// TwinCAT 3 PLC project PLC1
// Title: Sample Demo-Rack
// Company: Beckhoff Automation GmbH & Co. KG
// Author: Michael Golz
// ProjectVersion: 1.0.0
// ProgramVersion: 3.1.4026.26
// libraries:
//   Standard, * (System)
//   Tc2_Drive, * (Beckhoff Automation GmbH)
//   Tc2_EtherCAT, * (Beckhoff Automation GmbH)
//   Tc2_IoFunctions, * (Beckhoff Automation GmbH)
//   Tc2_Math, * (Beckhoff Automation GmbH)
//   Tc2_MC2, * (Beckhoff Automation GmbH)
//   Tc2_MC2_Camming, * (Beckhoff Automation GmbH)
//   Tc2_MC2_Drive, * (Beckhoff Automation GmbH)
//   Tc2_MC2_XFC, * (Beckhoff Automation GmbH)
//   Tc2_NCI, * (Beckhoff Automation GmbH)
//   Tc2_NcKinematicTransformation, * (Beckhoff Automation GmbH)
//   Tc2_PlcInterpolation, * (Beckhoff Automation GmbH)
//   Tc2_Standard, * (Beckhoff Automation GmbH)
//   Tc2_SUPS, * (Beckhoff Automation GmbH)
//   Tc2_System, * (Beckhoff Automation GmbH)
//   Tc2_Utilities, * (Beckhoff Automation GmbH)
//   Tc3_Database, * (Beckhoff Automation GmbH)
//   Tc3_EventLogger, * (Beckhoff Automation GmbH)
//   Tc3_Interfaces, * (Beckhoff Automation GmbH)
//   Tc3_IotBase, * (Beckhoff Automation GmbH)
//   Tc3_JsonXml, * (Beckhoff Automation GmbH)
//   Tc3_Mc3Base, * (Beckhoff Automation GmbH)
//   Tc3_Mc3FluidPower, * (Beckhoff Automation GmbH)
//   Tc3_Mc3Ptp, * (Beckhoff Automation GmbH)
//   Tc3_Module, * (Beckhoff Automation GmbH)
//   Tc3_RealtimeMonitoring, * (Beckhoff Automation GmbH)
//   TwinSafe3Diagnostics_v0.2.3, * (Beckhoff Automation LLC - Sample Code)
//   VisuDialogs, * (System)
// project tree:
//   DUTs/00_MainBlocks/ E_SystemStartupSequence.TcDUT (not stored)
//   DUTs/20_Axis/ E_AxisReversingSequence.TcDUT (not stored), E_McResetStatus.TcDUT (not stored)
//   DUTs/30_EtherCatDiagnostic/ E_EcDiacStatus.TcDUT (not stored), E_EcGetSlaveName.TcDUT (not stored), E_EcSystemStatus.TcDUT (not stored), ST_EcTerminalDiagInfo.TcDUT (not stored)
//   DUTs/40_TwinSAFE/ ST_AdsAddr.TcDUT (not stored)
//   DUTs/40_TwinSAFE/TwinSAFE_Connection/AX5805/ E_TsDiagnosisObjektsFA10AX5805.TcDUT (not stored), E_TsErrIndicesFA82AX5805.TcDUT (not stored), ST_TsControlWordAX5805.TcDUT (not stored), ST_TsDiagObjectsFA10AX5805.TcDUT (not stored), ST_TsErrIndicesFA82AX5805.TcDUT (not stored), ST_TsStatusWordAX5805.TcDUT (not stored)
//   DUTs/40_TwinSAFE/TwinSAFE_Connection/EK1914/ ST_TsDiagObjectsBitsEK1914.TcDUT (not stored), ST_TsDiagObjectsEK1914.TcDUT (not stored)
//   DUTs/40_TwinSAFE/TwinSAFE_Connection/EL1904/ ST_TsDiagObjectsBitsEL1904.TcDUT (not stored), ST_TsDiagObjectsEL1904.TcDUT (not stored)
//   DUTs/40_TwinSAFE/TwinSAFE_Connection/EL2904/ ST_TsDiagObjectsBitsEL2904.TcDUT (not stored), ST_TsDiagObjectsEL2904.TcDUT (not stored)
//   DUTs/40_TwinSAFE/TwinSAFE_Connection/ E_TsCycleDiagObj.TcDUT (not stored), ST_TsConnectionInfo1Byte.TcDUT (not stored), ST_TsConnectionInfo2Byte.TcDUT (not stored), ST_TsConnectionInfo8Byte.TcDUT (not stored), ST_TsConnectionInfoEL3214.TcDUT (not stored), ST_TsConnectionInfoEL5021.TcDUT (not stored), ST_TsSlave2Temp.TcDUT (not stored), ST_TsSlave3Temp.TcDUT (not stored)
//   DUTs/40_TwinSAFE/TwinSAFE_Functionblocks/ E_TsFbType.TcDUT (not stored), ST_TsFbInfo.TcDUT (not stored)
//   DUTs/40_TwinSAFE/TwinSAFE_Group/ ST_TsGroupInfo.TcDUT (not stored)
//   DUTs/ E_SampleMode.TcDUT (not stored)
//   / extMarkTask.TcTTO (not stored), FluidPowerSim.TcTTO, GlobalTextList.TcGTLO (not stored), NC_Task_1_SAF.TcTTO, PlcTask.TcTTO, PlcTaskFast.TcTTO (not stored), Visualization Manager.TcVMO (not stored)
//   GVLs/ GVL.TcGVL, GVL00_IO_CX.TcGVL (not stored), GVL01_IO_EK1100.TcGVL (not stored), GVL02_IO_EK1101.TcGVL (not stored), GVL10_VAR_PRG.TcGVL (not stored), GVL20_Axis.TcGVL, GVL30_DiagnosticEtherCAT.TcGVL (not stored)
//   POUs/MC3/ExternalSetpoint_Mc3_Nc2/ ExtSetpoint_MC3_NC2.TcPOU, FB_ExtSg_FollowNcAxis.TcPOU, PRG_SAF.TcPOU
//   POUs/MC3/ExternalSetpoint_Mc3_Nc2/Support/ E_Command.TcDUT, E_State.TcDUT
//   POUs/MC3/Gearing/ MC3_Gearing.TcPOU
//   POUs/MC3/Gearing/Support/ CompareLREAL.TcPOU, E_Axis.TcDUT, E_GearCommand.TcDUT, NextMinorStep.TcPOU (not stored), NextStep.TcPOU (not stored), SetStep.TcPOU
//   POUs/MC3/LoadControl/ LoadControl.TcPOU, LoadControlSim.TcPOU
//   POUs/MC3/PressToTarget/ PressToTarget.TcPOU, PressToTargetSim.TcPOU
//   POUs/MC3/ReversingSequence/ MC3_ReversingSequence.TcPOU
//   POUs/Motion/ CamTable.TcPOU (not stored), Ext_SP_Gen.TcPOU (not stored), Axis1.TcPOU, AxisGeneral.TcPOU (not stored), Axis2.TcPOU, Axis3.TcPOU, Axis4.TcPOU, NCI.TcPOU (not stored)
//   POUs/Database Server/ CSVSample.TcPOU (not stored), E_WriteMode.TcDUT (not stored), FB_CSV_Access.TcPOU (not stored), ST_CSVDataStruct.TcDUT (not stored)
//   POUs/GeneralPlcBlocks/ FB_GenerateData.TcPOU (not stored), Blinker.TcPOU (not stored), ClockGenerator.TcPOU (not stored), GeneralPlc.TcPOU (not stored)
//   POUs/IoT and JsonXml/FBs/ FB_JSONEncoding.TcPOU (not stored), FB_MqttCom_String.TcPOU (not stored), prgPopulateStructure.TcPOU (not stored)
//   POUs/IoT and JsonXml/ IoTDataStruct.TcDUT (not stored), IoT_JSON_XML.TcPOU (not stored)
//   POUs/MainPOUs/ MAIN.TcPOU, MAINFast.TcPOU (not stored), V_MAIN.TcVIS (not stored)
//   POUs/GeneralPlcBlocks/Components/ FB_Blinker.TcPOU (not stored), F_Scaling.TcPOU (not stored)
//   POUs/Motion/Components/ FB_Axis.TcPOU, FB_AxisAX5xxx.TcPOU, FB_ReversingSequence.TcPOU, MC_Reset_Ax5xxx.TcPOU
//   POUs/EtherCatDiagnostic/Components/ FB_DiagnosticEtherCAT.TcPOU (not stored)
//   POUs/EtherCatDiagnostic/ DiagnosticEtherCAT.TcPOU (not stored)
//   POUs/RT Monitor/ extMarksPrg.TcPOU (not stored), simpleMarksPrg.TcPOU (not stored)
//   POUs/RT Monitor/logging/ ConsumeTime.TcPOU (not stored)
//   POUs/Sample OOP/Cylinder/ FB_Cylinder.TcPOU (not stored), FB_CylinderDiag.TcPOU (not stored), ICylinder.TcIO (not stored)
//   POUs/Sample OOP/ FB_OOPAxisTable.TcPOU, FB_OOPCylinderRegulator.TcPOU (not stored)
//   POUs/Sample OOP/Regulator/ FB_BasicP.TcPOU (not stored), FB_BasicPID.TcPOU (not stored), IRegulator.TcIO (not stored), ST_RegParams.TcDUT (not stored)
//   POUs/Sample OOP/Table/Axis/ FB_AX5000Axis.TcPOU (not stored), FB_NcAxis.TcPOU, IAxis.TcIO (not stored)
//   POUs/Sample OOP/Table/ E_AxisState.TcDUT (not stored), E_MoveCmd.TcDUT (not stored), FB_Table.TcPOU (not stored)
//   POUs/TwinSAFE/Components/ FB_EcGetSlaveName.TcPOU (not stored), FB_TwinSafeConnectionAX5805.TcPOU (not stored), FB_TwinSafeConnectionEK1914.TcPOU (not stored), FB_TwinSafeConnectionEL1904.TcPOU (not stored), FB_TwinSafeConnectionEL2904.TcPOU (not stored), FB_TwinSafeConnectionEL3214.TcPOU (not stored), FB_TwinSafeConnectionEL5021.TcPOU (not stored), FB_TwinSafeFB.TcPOU (not stored), FB_TwinSafeGroup.TcPOU (not stored), FB_TwinSafeGroupExt.TcPOU (not stored)
//   POUs/TwinSAFE/ TwinSAFE.TcPOU (not stored)
//   POUs/XFC/ AverageOut.TcPOU (not stored), DcTimes.TcPOU (not stored), AnalogOutputOversampling.TcPOU (not stored), PositionCamTimeStampAxis2.TcPOU (not stored), SignalLengthMeasurementCamAxis2.TcPOU (not stored), TouchProbeTimeStampCamAxis2.TcPOU (not stored)
//   POUs/Sample OOP Conveyor/Axis Blocks/ FB_AX5000.TcPOU (not stored), FB_AxisNc.TcPOU, FB_Stepper.TcPOU (not stored), FB_VeryBasicMotor.TcPOU (not stored), I_Axis.TcIO (not stored)
//   POUs/Sample OOP Conveyor/Device And Station Blocks/ FB_Conveyor.TcPOU (not stored), FB_Device.TcPOU (not stored), FB_Station.TcPOU (not stored), FB_TransferStation.TcPOU (not stored), GVL_Products.TcGVL (not stored), I_Mode.TcIO (not stored)
//   POUs/Sample OOP Conveyor/Device And Station Blocks/Internal/ E_Modes.TcDUT (not stored), E_PartQuality.TcDUT (not stored), ST_PartData.TcDUT (not stored)
//   POUs/Sample OOP Conveyor/ FB_OOPConveyor.TcPOU, V_OOP_Conveyor.TcVIS (not stored)
//   POUs/Sample OOP Conveyor/Internal Visus/ Conveyor.TcVIS (not stored), ConveyorAuto.TcVIS (not stored), ConveyorData.TcVIS (not stored)
//   POUs/Sample UML SC/ FB_UML_SC_Composite.TcPOU (not stored), FB_UML_SC_Lamp.TcPOU (not stored), GVL_UML.TcGVL (not stored), Visu_Composite.TcVIS (not stored), Visu_Lamp.TcVIS (not stored)
//   POUs/SampleIEC Languages/Datatypes/ E_Commands.TcDUT (not stored), E_Operation.TcDUT (not stored)
//   POUs/SampleIEC Languages/FunctionBlocks/ FB_CFC_SamplePOU.TcPOU (not stored), FB_CFC_SamplePouPageOriented.TcPOU (not stored), FB_FBD_IL_LD_SamplePOU.TcPOU (not stored), FB_SFC_SamplePou.TcPOU (not stored), FB_ST_SamplePOU.TcPOU (not stored)
//   POUs/SampleIEC Languages/ MAIN_CFC.TcPOU (not stored), MAIN_CFC_PageOriented.TcPOU (not stored), MAIN_FBD_IL_LD.TcPOU (not stored), MAIN_SFC.TcPOU (not stored), MAIN_ST.TcPOU (not stored)
//   VISUs/ MotionProfiles.TcVIS (not stored), HmiEtherCatDiagnostic.TcVIS (not stored), HmiAxisReversingSequence.TcVIS (not stored), HmiStartPage.TcVIS (not stored), HmiTwinSAFEDiagnostic.TcVIS (not stored)
//   VISUs/HmiTemplatesAxis/ TplAxisControl.TcVIS (not stored), TplAxisReversingSequence.TcVIS (not stored)
//   VISUs/HmiTemplatesTwinSAFE/ TplTsConnectionAX5805.TcVIS (not stored), TplTsConnectionEK1914.TcVIS (not stored), TplTsConnectionEL1904.TcVIS (not stored), TplTsConnectionEL2904.TcVIS (not stored), TplTsConnectionEL3214.TcVIS (not stored), TplTsConnectionEL5021.TcVIS (not stored), TplTsFb.TcVIS (not stored), TplTsGroup.TcVIS (not stored), TplTsGroupExt.TcVIS (not stored)
// real-time tasks:
//   TASK PlcTask: cycle T#1ms, priority 8, ADS port 350
//   TASK PlcTaskFast: cycle T#100us, priority 4, ADS port 351
//   TASK VISU_TASK: cycle T#200000us, priority 30, ADS port 352
//   TASK extMarkTask: cycle T#1ms, priority 20, ADS port 353
//   TASK Job Task: cycle default, priority 32
//   TASK MC-Task (MET): cycle T#2ms, priority 14, ADS port 521
//   TASK MC-Task (MPT): cycle T#10ms, priority 15, ADS port 531
//   TASK FluidPowerSim: cycle T#2ms, priority 16, ADS port 354
// motion (NC):
//   TASK NC-Task 1 SAF: cycle T#1ms, priority 6, ADS port 501
//   TASK NC-Task 1 SVB: cycle T#10ms, priority 12, ADS port 511
//   AXIS Axis 1 Stepper (id 1)
//     General: UnitName=Degree
//     Dynamic: Acceleration=21600, Deceleration=21600, Jerk=259200, DelayTime=0.004
//     Velo: SlowManual=10, FastManual=150, Maximum=3600
//     OtherSettings: AllowMotionCmdToSlave=true
//     encoder EncType=4
//       EncPara: ScaleFactorNumerator=0.087890625, Inverse=true, EncMode=3, MaxCount=#xffffffff
//         Inc: RefSoftSyncMask=#x0000ffff
//     drive DrvType=24
//       DrvPara: Inverse=true
//         Analog: VeloReferenz=3600
//         TimeComp: TaskDelayCycles=1
//     controller CtrType=1
//       CtrPara: PriorControlFactor=1
//         PosDiffControl: Range=10
//         PID: PosKp=70
//         Observer: BandWidth=20
//   AXIS Axis 2 Servo EL (id 2)
//     Dynamic: Acceleration=5154.753, Deceleration=5154.753, Jerk=15464.259, DelayTime=0.004
//     Velo: RefSearch=34.36502, RefSync=34.36502, SlowManual=171.8251, FastManual=1030.9506, Fast=3436.502, Maximum=3436.502
//     OtherSettings: AllowMotionCmdToSlave=true
//     encoder EncType=19
//       EncPara: ScaleFactorNumerator=104.8576, ScaleFactorDenominator=1048576, Offset=-47.46, EncMode=3, MaxCount=#xffffffff
//     drive DrvType=16
//       DrvPara: MaxCount=#xffffffff, DriveControlDWord=#x00000100
//         Analog: VeloReferenz=3780.1522, VeloScale=32
//         TimeComp: TaskDelayCycles=1
//     controller CtrType=1
//       CtrPara: PriorControlFactor=1
//         PosDiffControl: Range=10
//         PID: PosKp=40
//         Observer: BandWidth=20
//   AXIS Axis 3 Servo A AX (id 3)
//     General: UnitName=Degree
//     Dynamic: Acceleration=108000, Deceleration=108000, Jerk=1296000
//     Velo: RefSearch=180, RefSync=180, SlowManual=10, FastManual=150, Fast=18000, Maximum=18000
//     OtherSettings: AllowMotionCmdToSlave=true
//     encoder EncType=8
//       EncPara: ScaleFactorNumerator=360, ScaleFactorDenominator=1048576, Offset=267.17, Inverse=true, MaxCount=#xffffffff
//     drive DrvType=9
//       DrvPara: Inverse=true, MaxCount=#xffffffff, DriveControlDWord=#x00030100
//         Analog: VeloReferenz=19800, VeloScale=1.02400649589962
//         TimeComp: TaskDelayCycles=1
//     controller CtrType=1
//       CtrPara: PriorControlFactor=1
//         PosDiffControl: Enable=false
//         Observer: BandWidth=20
//   AXIS Axis 4 Servo B AX (id 4)
//     General: UnitName=Degree
//     Dynamic: Acceleration=270000, Deceleration=270000, Jerk=8100000
//     Velo: RefSearch=180, RefSync=180, SlowManual=10, FastManual=150, Fast=18000, Maximum=18000
//     OtherSettings: AllowMotionCmdToSlave=true
//     encoder EncType=8
//       EncPara: ScaleFactorNumerator=360, ScaleFactorDenominator=1048576, Offset=16.16, MaxCount=#xffffffff
//     drive DrvType=9
//       DrvPara: MaxCount=#xffffffff, DriveControlDWord=#x00030100
//         Analog: VeloReferenz=19800, VeloScale=1.02400649589962
//         TimeComp: TaskDelayCycles=1
//     controller CtrType=1
//       CtrPara: PriorControlFactor=1
//         Observer: BandWidth=20
//   AXIS Axis 5 Handwheel (id 5)
//     OtherSettings: AllowMotionCmdToSlave=true
//     encoder EncType=4
//       EncPara: ScaleFactorNumerator=0.0375, Inverse=true, MaxCount=#x0000ffff
//         Inc: RefSoftSyncMask=#x0000ffff
//     drive DrvType=5
//       TimeComp: TaskDelayCycles=1
//     controller CtrType=1
//       CtrPara: PriorControlFactor=1
//         Observer: BandWidth=20
//   AXIS MC3_ExtMaster (id 6)
//     OtherSettings: AllowMotionCmdToSlave=true
//     encoder EncType=1
//     drive DrvType=5
//       Analog: TorqueSetpointScale=10, ScaleFactorActTorque=0.1
//       TimeComp: TaskDelayCycles=1
//     controller CtrType=1
//       CtrPara: PriorControlFactor=1
//         Observer: BandWidth=20
// I/O:
//   DEVICE Device 1 (EtherCAT), AmsNetId 169.254.108.162.2.1
//     Term 1 (EK1200) [EK1200-5000 EtherCAT Power supply (2A E-Bus)]
//       Term 2 (EL1008) [EL1008 8Ch. Dig. Input 24V, 3ms]
//       Term 3 (EL2008) [EL2008 8Ch. Dig. Output 24V, 0.5A]
//       Term 4 (EL5151) [EL5151 1Ch. Inc. Encoder]
//       Term 5 (EL9110) [EL9110 Power Supplier with LED (24V, Diagnostics)]
//       Term 6 (EL9576) [EL9576 Brake chopper terminal]
//       Term 7 (EL7037) [EL7037 1Ch. Stepper motor output stage (24V, 1.5A)]
//       Term 8 (EL9512) [EL9512 Power supply terminal 12V]
//       Term 9 (EL3162) [EL3162 2Ch. Ana. Input 0-10V]
//       Term 10 (EL4102) [EL4102 2Ch. Ana. Output  0-10V, 16bit]
//       Term 11 (EL6900) [EL6900, TwinSAFE PLC] (disabled)
//       Term 43 (EL6910) [EL6910, TwinSAFE PLC]
//       Term 12 (EK1122) [EK1122 2 port EtherCAT junction]
//         Drive 29 (AX5203-0000-0215)_1 [AX5203-0000-0215 EtherCAT Drive (SoE, 2 Ch.)]
//           Term 34 (AX5805) [AX5805 (Safety Drive Option)]
//             modules: Module 1 (Safety Process Data, 2 axis), Module 2 (Standard Process Data, 2 axis)
//         Term 13 (EK1100) [EK1100 EtherCAT Coupler (2A E-Bus)]
//           Term 14 (EL1859) [EL1859 8Ch. Dig. Input 24V, 3ms, 8Ch. Dig. Output 24V, 0.5A]
//           Term 15 (EL1904) [EL1904, 4 Ch. Safety Input 24V, TwinSAFE]
//             modules: Module 1 (FSOES)
//           Term 16 (EL2904) [EL2904, 4 Ch. Safety Output 24V, 0.5A, TwinSAFE]
//             modules: Module 1 (FSOES), Module 2 (DO)
//           Term 17 (EL9110) [EL9110 Power Supplier with LED (24V, Diagnostics)]
//           Term 18 (EL2004) [EL2004 4Ch. Dig. Output 24V, 0.5A]
//           Term 19 (EL9410) [EL9410 E-Bus Power Supplier  (Diagnostics)]
//           Term 20 (EL7201-0010) [EL7201-0010 1Ch. MDP742 Servo motor output stage with OCT (50V, 4A)]
//             startup 32784:18 := 0500
//             startup 32784:19 := B200
//             startup 32784:20 := 96000000 // Velocity loop integral time
//             startup 32784:21 := 2B000000 // Velocity loop proportional gain
//             startup 32785:17 := 98210000
//             startup 32785:18 := 960A0000
//             startup 32785:19 := 03
//             startup 32785:21 := 0E01
//             startup 32785:22 := 46000000
//             startup 32785:24 := 21000000
//             startup 32785:25 := 0F00
//             startup 32785:27 := 4F060000
//             startup 32785:45 := 5501
//           Term 30 (EL9011) [EL9011 End Terminal]
//     Term 21 (EK1101) [EK1101 EtherCAT Coupler (2A E-Bus, ID switch)]
//       Term 22 (EL1904) [EL1904, 4 Ch. Safety Input 24V, TwinSAFE]
//         modules: Module 1 (FSOES)
//       Term 23 (EL1252) [EL1252 2Ch. Fast Dig. Input 24V, 1µs, DC Latch]
//       Term 24 (EL1262) [EL1262 2Ch. Dig. Input 24V, 1µs, DC Oversample]
//       Term 25 (EL2252) [EL2252 2Ch. Dig. Output 24V, 0.5A, DC Time Stamp]
//       Term 26 (EL3702) [EL3702 2Ch. Ana. Input +/-10V, DIFF, Oversample]
//       Term 27 (EL4732) [EL4732 2Ch. Ana. Output +/-10V, Oversample]
//       Term 28 (EL2004) [EL2004 4Ch. Dig. Output 24V, 0.5A]
//       Term 31 (EL9011) [EL9011 End Terminal]
// variable links:
//   Device 1 (EtherCAT) <-> Device 1 (EtherCAT)/Term 1 (EK1200)/Term 12 (EK1122)/Drive 29 (AX5203-0000-0215)_1/Term 34 (AX5805)
//     Term 1 (EK1200)/Term 43 (EL6910)/ConnectionInputs/Message_5 TxPDO <-> Module 1 (Safety Process Data, 2 axis)/Outputs (Controlword)/FSOE
//     Term 1 (EK1200)/Term 43 (EL6910)/ConnectionOutputs/Message_5 RxPDO <-> Module 1 (Safety Process Data, 2 axis)/Inputs (Statusword)/FSOE
//   Device 1 (EtherCAT) <-> Device 1 (EtherCAT)/Term 1 (EK1200)/Term 12 (EK1122)/Term 13 (EK1100)/Term 15 (EL1904)
//     Term 1 (EK1200)/Term 43 (EL6910)/ConnectionInputs/Message_2 TxPDO <-> Module 1 (FSOES)/RxPDO/FSOE
//     Term 1 (EK1200)/Term 43 (EL6910)/ConnectionOutputs/Message_2 RxPDO <-> Module 1 (FSOES)/TxPDO/FSOE
//   Device 1 (EtherCAT) <-> Device 1 (EtherCAT)/Term 1 (EK1200)/Term 12 (EK1122)/Term 13 (EK1100)/Term 16 (EL2904)
//     Term 1 (EK1200)/Term 43 (EL6910)/ConnectionInputs/Message_3 TxPDO <-> Module 1 (FSOES)/RxPDO/FSOE
//     Term 1 (EK1200)/Term 43 (EL6910)/ConnectionOutputs/Message_3 RxPDO <-> Module 1 (FSOES)/TxPDO/FSOE
//   Device 1 (EtherCAT) <-> Device 1 (EtherCAT)/Term 21 (EK1101)/Term 22 (EL1904)
//     Term 1 (EK1200)/Term 43 (EL6910)/ConnectionInputs/Message_4 TxPDO <-> Module 1 (FSOES)/RxPDO/FSOE
//     Term 1 (EK1200)/Term 43 (EL6910)/ConnectionOutputs/Message_4 RxPDO <-> Module 1 (FSOES)/TxPDO/FSOE
//   NC-Task 1 SAF/Axes/Axis 1 Stepper <-> Device 1 (EtherCAT)/Term 1 (EK1200)/Term 7 (EL7037)
//     Drive/Inputs/In/nState1 @bit 3 <-> STM Status/Status/Error
//     Drive/Inputs/In/nState1 @bit 7 <-> STM Status/Status/Motor stall
//     Drive/Inputs/In/nState1 @bit 5 <-> STM Status/Status/Moving negative
//     Drive/Inputs/In/nState1 @bit 4 <-> STM Status/Status/Moving positive
//     Drive/Inputs/In/nState1 @bit 1 <-> STM Status/Status/Ready
//     Drive/Inputs/In/nState1 <-> STM Status/Status/Ready to enable
//     Drive/Inputs/In/nState1 @bit 6 <-> STM Status/Status/Torque reduced
//     Drive/Inputs/In/nState1 @bit 2 <-> STM Status/Status/Warning
//     Drive/Inputs/In/nState2 @bit 3 <-> STM Status/Status/Digital input 1
//     Drive/Inputs/In/nState2 @bit 4 <-> STM Status/Status/Digital input 2
//     Drive/Inputs/In/nState2 @bit 5 <-> STM Status/Status/Sync error
//     Drive/Inputs/In/nState2 @bit 7 <-> STM Status/Status/TxPDO Toggle
//     Drive/Inputs/In/nState4 @bit 1 <-> WcState/InputToggle
//     Drive/Inputs/In/nState4 <-> WcState/WcState
//     Drive/Outputs/Out/nCtrl1 <-> STM Control/Control/Enable
//     Drive/Outputs/Out/nCtrl1 @bit 2 <-> STM Control/Control/Reduce torque
//     Drive/Outputs/Out/nCtrl1 @bit 1 <-> STM Control/Control/Reset
//     Drive/Outputs/Out/nCtrl2 @bit 3 <-> STM Control/Control/Digital output 1
//     Drive/Outputs/Out/nDataOut2[0] <-> STM Velocity/Velocity
//     Enc/Inputs/In/nDataIn1 <-> ENC Status/Counter value
//     Enc/Inputs/In/nDataIn2 <-> ENC Status/Latch value
//     Enc/Inputs/In/nState1 @bit 4 <-> ENC Status/Status/Counter overflow
//     Enc/Inputs/In/nState1 @bit 3 <-> ENC Status/Status/Counter underflow
//     Enc/Inputs/In/nState1 @bit 7 <-> ENC Status/Status/Extrapolation stall
//     Enc/Inputs/In/nState1 <-> ENC Status/Status/Latch C valid
//     Enc/Inputs/In/nState1 @bit 1 <-> ENC Status/Status/Latch extern valid
//     Enc/Inputs/In/nState1 @bit 2 <-> ENC Status/Status/Set counter done
//     Enc/Inputs/In/nState2 @bit 4 <-> ENC Status/Status/Status of extern latch
//     Enc/Inputs/In/nState2 <-> ENC Status/Status/Status of input A
//     Enc/Inputs/In/nState2 @bit 1 <-> ENC Status/Status/Status of input B
//     Enc/Inputs/In/nState2 @bit 2 <-> ENC Status/Status/Status of input C
//     Enc/Inputs/In/nState2 @bit 5 <-> ENC Status/Status/Sync error
//     Enc/Inputs/In/nState2 @bit 7 <-> ENC Status/Status/TxPDO Toggle
//     Enc/Inputs/In/nState4 @bit 1 <-> WcState/InputToggle
//     Enc/Inputs/In/nState4 <-> WcState/WcState
//     Enc/Outputs/Out/nCtrl1 <-> ENC Control/Control/Enable latch C
//     Enc/Outputs/Out/nCtrl1 @bit 3 <-> ENC Control/Control/Enable latch extern on negative edge
//     Enc/Outputs/Out/nCtrl1 @bit 1 <-> ENC Control/Control/Enable latch extern on positive edge
//     Enc/Outputs/Out/nCtrl1 @bit 2 <-> ENC Control/Control/Set counter
//     Enc/Outputs/Out/nDataOut1 <-> ENC Control/Set counter value
//   NC-Task 1 SAF/Axes/Axis 2 Servo EL <-> Device 1 (EtherCAT)/Term 1 (EK1200)/Term 12 (EK1122)/Term 13 (EK1100)/Term 20 (EL7201-0010)
//     Drive/Inputs/In/nDataIn1 <-> DRV Following error actual value/Following error actual value
//     Drive/Inputs/In/nDataIn3[0] <-> DRV Torque actual value/Torque actual value
//     Drive/Inputs/In/nDcOutputTime <-> InfoData/DcOutputShift
//     Drive/Inputs/In/nState1 <-> DRV Statusword/Statusword
//     Drive/Inputs/In/nState2 <-> DRV Statusword/Statusword @bit 8
//     Drive/Inputs/In/nState4 @bit 1 <-> WcState/InputToggle
//     Drive/Inputs/In/nState4 <-> WcState/WcState
//     Drive/Outputs/Out/nCtrl1 <-> DRV Controlword/Controlword
//     Drive/Outputs/Out/nCtrl2 <-> DRV Controlword/Controlword @bit 8
//     Drive/Outputs/Out/nDataOut1 <-> DRV Target position/Target position
//     Drive/Outputs/Out/nDataOut2 <-> DRV Target velocity/Target velocity
//     Enc/Inputs/In/nDataIn1 <-> FB Position/Position
//     Enc/Inputs/In/nDcInputTime <-> InfoData/DcInputShift
//     Enc/Inputs/In/nState4 @bit 1 <-> WcState/InputToggle
//     Enc/Inputs/In/nState4 <-> WcState/WcState
//     Enc/Inputs/In/nState5 <-> FB Touch probe status/Touch probe status/TP1 Enable
//     Enc/Inputs/In/nState6 <-> FB Touch probe status/Touch probe status/TP2 Enable
//     Enc/Inputs/In/nState5 @bit 7 <-> FB Touch probe status/Touch probe status/TP1 Input
//     Enc/Inputs/In/nState6 @bit 7 <-> FB Touch probe status/Touch probe status/TP2 Input
//     Enc/Inputs/In/nState5 @bit 2 <-> FB Touch probe status/Touch probe status/TP1 Neg value stored
//     Enc/Inputs/In/nState6 @bit 2 <-> FB Touch probe status/Touch probe status/TP2 Neg value stored
//     Enc/Inputs/In/nState5 @bit 1 <-> FB Touch probe status/Touch probe status/TP1 Pos value stored
//     Enc/Inputs/In/nState6 @bit 1 <-> FB Touch probe status/Touch probe status/TP2 Pos value stored
//   NC-Task 1 SAF/Axes/Axis 3 Servo A AX <-> Device 1 (EtherCAT)/Term 1 (EK1200)/Term 12 (EK1122)/Drive 29 (AX5203-0000-0215)_1
//     Drive/Inputs/In/nDataIn1 <-> AT 1/Following distance
//     Drive/Inputs/In/nDcOutputTime <-> InfoData/DcOutputShift
//     Drive/Inputs/In/nState1 <-> AT 1/Drive status word @bit 8
//     Drive/Inputs/In/nState2 <-> AT 1/Drive status word
//     Drive/Inputs/In/nState4 @bit 1 <-> WcState/InputToggle
//     Drive/Outputs/Out/nCtrl1 <-> MDT 1/Master control word @bit 8
//     Drive/Outputs/Out/nDataOut1 <-> MDT 1/Position command value
//     Enc/Inputs/In/nDataIn1 <-> AT 1/Position feedback 1 value
//     Enc/Inputs/In/nDcInputTime <-> InfoData/DcInputShift
//     Enc/Inputs/In/nState4 @bit 1 <-> WcState/InputToggle
//   NC-Task 1 SAF/Axes/Axis 4 Servo B AX <-> Device 1 (EtherCAT)/Term 1 (EK1200)/Term 12 (EK1122)/Drive 29 (AX5203-0000-0215)_1
//     Drive/Inputs/In/nDataIn1 <-> AT 2/Following distance
//     Drive/Inputs/In/nDcOutputTime <-> InfoData/DcOutputShift
//     Drive/Inputs/In/nState1 <-> AT 2/Drive status word @bit 8
//     Drive/Inputs/In/nState2 <-> AT 2/Drive status word
//     Drive/Inputs/In/nState4 @bit 1 <-> WcState/InputToggle
//     Drive/Outputs/Out/nCtrl1 <-> MDT 2/Master control word @bit 8
//     Drive/Outputs/Out/nDataOut1 <-> MDT 2/Position command value
//     Enc/Inputs/In/nDataIn1 <-> AT 2/Position feedback 1 value
//     Enc/Inputs/In/nDcInputTime <-> InfoData/DcInputShift
//     Enc/Inputs/In/nState4 @bit 1 <-> WcState/InputToggle
//   NC-Task 1 SAF/Axes/Axis 5 Handwheel <-> Device 1 (EtherCAT)/Term 1 (EK1200)/Term 4 (EL5151)
//     Enc/Inputs/In/nDataIn1[0] <-> ENC Inputs/Counter value
//     Enc/Inputs/In/nDataIn2[0] <-> ENC Inputs/Latch value
//     Enc/Inputs/In/nState1 @bit 7 <-> ENC Inputs/Status/Extrapolation stall
//     Enc/Inputs/In/nState1 <-> ENC Inputs/Status/Latch C valid
//     Enc/Inputs/In/nState1 @bit 1 <-> ENC Inputs/Status/Latch extern valid
//     Enc/Inputs/In/nState1 @bit 2 <-> ENC Inputs/Status/Set counter done
//     Enc/Inputs/In/nState2 @bit 4 <-> ENC Inputs/Status/Status of extern latch
//     Enc/Inputs/In/nState2 <-> ENC Inputs/Status/Status of input A
//     Enc/Inputs/In/nState2 @bit 1 <-> ENC Inputs/Status/Status of input B
//     Enc/Inputs/In/nState2 @bit 2 <-> ENC Inputs/Status/Status of input C
//     Enc/Inputs/In/nState2 @bit 5 <-> ENC Inputs/Status/Sync error
//     Enc/Inputs/In/nState2 @bit 7 <-> ENC Inputs/Status/TxPDO Toggle
//     Enc/Inputs/In/nState4 @bit 1 <-> WcState/InputToggle
//     Enc/Inputs/In/nState4 <-> WcState/WcState
//     Enc/Outputs/Out/nCtrl1 <-> ENC Outputs/Control/Enable latch C
//     Enc/Outputs/Out/nCtrl1 @bit 3 <-> ENC Outputs/Control/Enable latch extern on negative edge
//     Enc/Outputs/Out/nCtrl1 @bit 1 <-> ENC Outputs/Control/Enable latch extern on positive edge
//     Enc/Outputs/Out/nCtrl1 @bit 2 <-> ENC Outputs/Control/Set counter
//     Enc/Outputs/Out/nDataOut1[0] <-> ENC Outputs/Set counter value
//   PLC1/PLC1 Instance <-> Device 1 (EtherCAT)
//     PlcTask Inputs/GVL30_DiagnosticEtherCAT.fbDiagnosticEtherCAT.cbAmsNetId <-> InfoData/AmsNetId
//     PlcTask Inputs/GVL30_DiagnosticEtherCAT.fbDiagnosticEtherCAT.nCfgSlaveCount <-> InfoData/CfgSlaveCount
//     PlcTask Inputs/GVL30_DiagnosticEtherCAT.fbDiagnosticEtherCAT.nDevId <-> InfoData/DevId
//     PlcTask Inputs/GVL30_DiagnosticEtherCAT.fbDiagnosticEtherCAT.nDevState <-> Inputs/DevState
//     PlcTask Inputs/GVL30_DiagnosticEtherCAT.fbDiagnosticEtherCAT.nFrmXWcState[0] <-> Inputs/Frm0WcState
//   PLC1/PLC1 Instance <-> Device 1 (EtherCAT)/Term 1 (EK1200)/Term 10 (EL4102)
//     PlcTask Outputs/GVL00_IO_CX.nAnalogOutP10 <-> Channel 1/Output
//     PlcTaskFast Outputs/GVL00_IO_CX.nAnalogOutP11 <-> Channel 2/Output
//   PLC1/PLC1 Instance <-> Device 1 (EtherCAT)/Term 1 (EK1200)/Term 12 (EK1122)/Drive 29 (AX5203-0000-0215)_1
//     PlcTask Inputs/GVL20_Axis.nAX5203DigitalInputs <-> AT 1/Digital inputs, state
//     PlcTask Inputs/GVL20_Axis.nAxis3TorqueFeedback <-> AT 1/Torque/force feedback value
//     PlcTask Inputs/GVL20_Axis.nAxis4TorqueFeedback <-> AT 2/Torque/force feedback value
//     PlcTask Outputs/GVL20_Axis.nAX5203DigitalOutputs <-> MDT 1/Digital outputs
//   PLC1/PLC1 Instance <-> Device 1 (EtherCAT)/Term 1 (EK1200)/Term 12 (EK1122)/Term 13 (EK1100)/Term 14 (EL1859)
//     PlcTask Inputs/GVL01_IO_EK1100.bAxis2ReferenceCamEL1 <-> Channel 5/Input
//     PlcTask Inputs/GVL01_IO_EK1100.bSwitchS20 <-> Channel 1/Input
//     PlcTask Inputs/GVL01_IO_EK1100.bSwitchS21 <-> Channel 2/Input
//     PlcTask Inputs/GVL01_IO_EK1100.bSwitchS22 <-> Channel 3/Input
//     PlcTask Inputs/GVL01_IO_EK1100.bSwitchS31 <-> Channel 4/Input
//     PlcTask Outputs/GVL01_IO_EK1100.bLedH23 <-> Channel 13/Output
//     PlcTask Outputs/GVL01_IO_EK1100.bLedH24 <-> Channel 14/Output
//     PlcTask Outputs/GVL01_IO_EK1100.bLedH25 <-> Channel 15/Output
//     PlcTask Outputs/GVL01_IO_EK1100.bLedH26 <-> Channel 16/Output
//     PlcTask Outputs/GVL01_IO_EK1100.bLedH31 <-> Channel 9/Output
//     PlcTask Outputs/GVL01_IO_EK1100.bLedH32 <-> Channel 10/Output
//     PlcTask Outputs/GVL01_IO_EK1100.bLedH33 <-> Channel 11/Output
//   PLC1/PLC1 Instance <-> Device 1 (EtherCAT)/Term 1 (EK1200)/Term 12 (EK1122)/Term 13 (EK1100)/Term 15 (EL1904)
//     PlcTask Inputs/TwinSAFE.fbSafeConnectionEL1904_1_Group1.nEcSlaveState <-> InfoData/State
//     PlcTask Inputs/TwinSAFE.fbSafeConnectionEL1904_1_Group1.stEcAdsAddr <-> InfoData/AdsAddr
//   PLC1/PLC1 Instance <-> Device 1 (EtherCAT)/Term 1 (EK1200)/Term 12 (EK1122)/Term 13 (EK1100)/Term 16 (EL2904)
//     PlcTask Inputs/TwinSAFE.fbSafeConnectionEL2904_1_Group1.nEcSlaveState <-> InfoData/State
//     PlcTask Inputs/TwinSAFE.fbSafeConnectionEL2904_1_Group1.stEcAdsAddr <-> InfoData/AdsAddr
//   PLC1/PLC1 Instance <-> Device 1 (EtherCAT)/Term 1 (EK1200)/Term 12 (EK1122)/Term 13 (EK1100)/Term 17 (EL9110)
//     PlcTask Inputs/GVL01_IO_EK1100.bPotentialConduktorK124VOk <-> PowerOK/Input
//   PLC1/PLC1 Instance <-> Device 1 (EtherCAT)/Term 1 (EK1200)/Term 12 (EK1122)/Term 13 (EK1100)/Term 18 (EL2004)
//     PlcTask Outputs/GVL01_IO_EK1100.bLedH20 <-> Channel 1/Output
//     PlcTask Outputs/GVL01_IO_EK1100.bLedH21 <-> Channel 2/Output
//     PlcTask Outputs/GVL01_IO_EK1100.bLedH22 <-> Channel 3/Output
//   PLC1/PLC1 Instance <-> Device 1 (EtherCAT)/Term 1 (EK1200)/Term 12 (EK1122)/Term 13 (EK1100)/Term 19 (EL9410)
//     PlcTask Inputs/GVL01_IO_EK1100.bPotentialEBusUs24VNotOk <-> Status Us/Undervoltage
//     PlcTask Inputs/GVL01_IO_EK1100.bPotentialServoUp24VNotOk <-> Status Up/Undervoltage
//   PLC1/PLC1 Instance <-> Device 1 (EtherCAT)/Term 1 (EK1200)/Term 2 (EL1008)
//     PlcTask Inputs/GVL00_IO_CX.bSwitchS10 <-> Channel 1/Input
//     PlcTask Inputs/GVL00_IO_CX.bSwitchS11 <-> Channel 2/Input
//     PlcTask Inputs/GVL00_IO_CX.bSwitchS12 <-> Channel 3/Input
//     PlcTask Inputs/GVL00_IO_CX.bSwitchS13 <-> Channel 4/Input
//     PlcTask Inputs/GVL00_IO_CX.bSwitchS14 <-> Channel 5/Input
//     PlcTask Inputs/GVL00_IO_CX.bSwitchS15 <-> Channel 6/Input
//     PlcTask Inputs/GVL00_IO_CX.bSwitchS16 <-> Channel 7/Input
//     PlcTask Inputs/GVL00_IO_CX.bSwitchS17 <-> Channel 8/Input
//   PLC1/PLC1 Instance <-> Device 1 (EtherCAT)/Term 1 (EK1200)/Term 3 (EL2008)
//     PlcTask Outputs/GVL00_IO_CX.bLedH10 <-> Channel 1/Output
//     PlcTask Outputs/GVL00_IO_CX.bLedH11 <-> Channel 2/Output
//     PlcTask Outputs/GVL00_IO_CX.bLedH12 <-> Channel 3/Output
//     PlcTask Outputs/GVL00_IO_CX.bLedH13 <-> Channel 4/Output
//     PlcTask Outputs/GVL00_IO_CX.bLedH14 <-> Channel 5/Output
//     PlcTask Outputs/GVL00_IO_CX.bLedH15 <-> Channel 6/Output
//     PlcTask Outputs/GVL00_IO_CX.bLedH16 <-> Channel 7/Output
//     PlcTask Outputs/GVL00_IO_CX.bLedH17 <-> Channel 8/Output
//   PLC1/PLC1 Instance <-> Device 1 (EtherCAT)/Term 1 (EK1200)/Term 4 (EL5151)
//     PlcTask Inputs/GVL00_IO_CX.bHandwheelSwitchS28 <-> ENC Inputs/Status/Status of extern latch
//     PlcTask Inputs/GVL00_IO_CX.nHandwheelCounter <-> ENC Inputs/Counter value
//   PLC1/PLC1 Instance <-> Device 1 (EtherCAT)/Term 1 (EK1200)/Term 43 (EL6910)
//     PlcTask Inputs/TwinSAFE.fbSafeGroup1.bComErr <-> StandardInputs/Standard Out Var 6
//     PlcTask Inputs/TwinSAFE.fbSafeGroup1.bFbErr <-> StandardInputs/Standard Out Var 7
//     PlcTask Inputs/TwinSAFE.fbSafeGroup1.bOutErr <-> StandardInputs/Standard Out Var 8
//     PlcTask Outputs/TwinSAFE.fbSafeGroup1.bErrAck <-> StandardOutputs/Standard In Var 1
//     PlcTask Outputs/TwinSAFE.fbSafeGroup1.bRun <-> StandardOutputs/Standard In Var 9
//   PLC1/PLC1 Instance <-> Device 1 (EtherCAT)/Term 1 (EK1200)/Term 5 (EL9110)
//     PlcTask Inputs/GVL00_IO_CX.bPotentialStepper24VOk <-> PowerOK/Input
//   PLC1/PLC1 Instance <-> Device 1 (EtherCAT)/Term 1 (EK1200)/Term 7 (EL7037)
//     PlcTask Inputs/GVL00_IO_CX.bStepperReferenceCam <-> ENC Status/Status/Status of extern latch
//     PlcTask Inputs/GVL00_IO_CX.bSwitchS23 <-> STM Status/Status/Digital input 1
//     PlcTask Inputs/GVL00_IO_CX.bSwitchS24 <-> STM Status/Status/Digital input 2
//   PLC1/PLC1 Instance <-> Device 1 (EtherCAT)/Term 1 (EK1200)/Term 8 (EL9512)
//     PlcTask Inputs/GVL00_IO_CX.bPotentialAnalog12VOk <-> Status Uo/Power OK
//   PLC1/PLC1 Instance <-> Device 1 (EtherCAT)/Term 1 (EK1200)/Term 9 (EL3162)
//     PlcTask Inputs/GVL00_IO_CX.nAnalogInFromEL4102Out1 <-> AI Standard Channel 2/Value
//     PlcTask Inputs/GVL00_IO_CX.nAnalogInR10 <-> AI Standard Channel 1/Value
//   PLC1/PLC1 Instance <-> Device 1 (EtherCAT)/Term 21 (EK1101)/Term 22 (EL1904)
//     PlcTask Inputs/TwinSAFE.fbSafeConnectionEL1904_2_Group1.nEcSlaveState <-> InfoData/State
//     PlcTask Inputs/TwinSAFE.fbSafeConnectionEL1904_2_Group1.stEcAdsAddr <-> InfoData/AdsAddr
//   PLC1/PLC1 Instance <-> Device 1 (EtherCAT)/Term 21 (EK1101)/Term 23 (EL1252)
//     PlcTask Inputs/GVL02_IO_EK1101.stEL1252Ch1.Input <-> Channel 1/Input
//     PlcTask Inputs/GVL02_IO_EK1101.stEL1252Ch2.Input <-> Channel 2/Input
//     PlcTask Inputs/GVL02_IO_EK1101.stEL1252Ch1.Status <-> Latch/Status1
//     PlcTask Inputs/GVL02_IO_EK1101.stEL1252Ch2.Status <-> Latch/Status2
//     PlcTask Inputs/GVL02_IO_EK1101.stEL1252Ch1.TimeStampNeg <-> Latch/LatchNeg1
//     PlcTask Inputs/GVL02_IO_EK1101.stEL1252Ch2.TimeStampNeg <-> Latch/LatchNeg2
//     PlcTask Inputs/GVL02_IO_EK1101.stEL1252Ch1.TimeStampPos <-> Latch/LatchPos1
//     PlcTask Inputs/GVL02_IO_EK1101.stEL1252Ch2.TimeStampPos <-> Latch/LatchPos2
//   PLC1/PLC1 Instance <-> Device 1 (EtherCAT)/Term 21 (EK1101)/Term 24 (EL1262)
//     PlcTask Inputs/GVL02_IO_EK1101.aAxis2RefCamOs[0] <-> Ch1 Input 0/Ch1 Input
//     PlcTask Inputs/GVL02_IO_EK1101.aAxis2RefCamOs[1] <-> Ch1 Input 1/Ch1 Input
//     PlcTask Inputs/GVL02_IO_EK1101.aAxis2RefCamOs[2] <-> Ch1 Input 2/Ch1 Input
//     PlcTask Inputs/GVL02_IO_EK1101.aAxis2RefCamOs[3] <-> Ch1 Input 3/Ch1 Input
//     PlcTask Inputs/GVL02_IO_EK1101.aAxis2RefCamOs[4] <-> Ch1 Input 4/Ch1 Input
//     PlcTask Inputs/GVL02_IO_EK1101.aAxis2RefCamOs[5] <-> Ch1 Input 5/Ch1 Input
//     PlcTask Inputs/GVL02_IO_EK1101.aAxis2RefCamOs[6] <-> Ch1 Input 6/Ch1 Input
//     PlcTask Inputs/GVL02_IO_EK1101.aAxis2RefCamOs[7] <-> Ch1 Input 7/Ch1 Input
//     PlcTask Inputs/GVL02_IO_EK1101.aAxis2RefCamOs[8] <-> Ch1 Input 8/Ch1 Input
//     PlcTask Inputs/GVL02_IO_EK1101.aAxis2RefCamOs[9] <-> Ch1 Input 9/Ch1 Input
//     PlcTask Inputs/GVL02_IO_EK1101.aOsInputFromEL2252Out2[0] <-> Ch2 Input 0/Ch2 Input
//     PlcTask Inputs/GVL02_IO_EK1101.aOsInputFromEL2252Out2[1] <-> Ch2 Input 1/Ch2 Input
//     PlcTask Inputs/GVL02_IO_EK1101.aOsInputFromEL2252Out2[2] <-> Ch2 Input 2/Ch2 Input
//     PlcTask Inputs/GVL02_IO_EK1101.aOsInputFromEL2252Out2[3] <-> Ch2 Input 3/Ch2 Input
//     PlcTask Inputs/GVL02_IO_EK1101.aOsInputFromEL2252Out2[4] <-> Ch2 Input 4/Ch2 Input
//     PlcTask Inputs/GVL02_IO_EK1101.aOsInputFromEL2252Out2[5] <-> Ch2 Input 5/Ch2 Input
//     PlcTask Inputs/GVL02_IO_EK1101.aOsInputFromEL2252Out2[6] <-> Ch2 Input 6/Ch2 Input
//     PlcTask Inputs/GVL02_IO_EK1101.aOsInputFromEL2252Out2[7] <-> Ch2 Input 7/Ch2 Input
//     PlcTask Inputs/GVL02_IO_EK1101.aOsInputFromEL2252Out2[8] <-> Ch2 Input 8/Ch2 Input
//     PlcTask Inputs/GVL02_IO_EK1101.aOsInputFromEL2252Out2[9] <-> Ch2 Input 9/Ch2 Input
//     PlcTask Inputs/GVL02_IO_EK1101.nEL1262Ch1CycleCount <-> Ch1 CycleCount/Ch1 CycleCount
//     PlcTask Inputs/GVL02_IO_EK1101.nEL1262Ch2CycleCount <-> Ch2 CycleCount/Ch2 CycleCount
//   PLC1/PLC1 Instance <-> Device 1 (EtherCAT)/Term 21 (EK1101)/Term 25 (EL2252)
//     PlcTask Outputs/GVL02_IO_EK1101.stEL2252.Activate <-> DC Sync Activate/Activate
//     PlcTask Outputs/GVL02_IO_EK1101.stEL2252.Output1 <-> Channel 1/Output
//     PlcTask Outputs/GVL02_IO_EK1101.stEL2252.Output2 <-> Channel 2/Output
//     PlcTask Outputs/GVL02_IO_EK1101.stEL2252.StartTime <-> DC Sync Start/StartTime
//     PlcTask Outputs/GVL02_IO_EK1101.stEL2252.TriState1 <-> Channel 1/TriState
//     PlcTask Outputs/GVL02_IO_EK1101.stEL2252.TriState2 <-> Channel 2/TriState
//   PLC1/PLC1 Instance <-> Device 1 (EtherCAT)/Term 21 (EK1101)/Term 26 (EL3702)
//     PlcTask Inputs/GVL02_IO_EK1101.nEL3702Ch1CycleCount <-> Ch1 CycleCount/Ch1 CycleCount
//     PlcTask Inputs/GVL02_IO_EK1101.nEL3702Ch2CycleCount <-> Ch2 CycleCount/Ch2 CycleCount
//     PlcTaskFast Inputs/GVL02_IO_EK1101.aOsAnalogInR11[0] <-> Ch1 Sample 0/Ch1 Value
//     PlcTaskFast Inputs/GVL02_IO_EK1101.aOsAnalogInR11[1] <-> Ch1 Sample 1/Ch1 Value
//     PlcTaskFast Inputs/GVL02_IO_EK1101.aOsAnalogInR11[2] <-> Ch1 Sample 2/Ch1 Value
//     PlcTaskFast Inputs/GVL02_IO_EK1101.aOsAnalogInR11[3] <-> Ch1 Sample 3/Ch1 Value
//     PlcTaskFast Inputs/GVL02_IO_EK1101.aOsAnalogInR11[4] <-> Ch1 Sample 4/Ch1 Value
//     PlcTaskFast Inputs/GVL02_IO_EK1101.aOsAnalogInR11[5] <-> Ch1 Sample 5/Ch1 Value
//     PlcTaskFast Inputs/GVL02_IO_EK1101.aOsAnalogInR11[6] <-> Ch1 Sample 6/Ch1 Value
//     PlcTaskFast Inputs/GVL02_IO_EK1101.aOsAnalogInR11[7] <-> Ch1 Sample 7/Ch1 Value
//     PlcTaskFast Inputs/GVL02_IO_EK1101.aOsAnalogInR11[8] <-> Ch1 Sample 8/Ch1 Value
//     PlcTaskFast Inputs/GVL02_IO_EK1101.aOsAnalogInR11[9] <-> Ch1 Sample 9/Ch1 Value
//     PlcTaskFast Inputs/GVL02_IO_EK1101.aOsInputFromEL4732Out1[0] <-> Ch2 Sample 0/Ch2 Value
//     PlcTaskFast Inputs/GVL02_IO_EK1101.aOsInputFromEL4732Out1[1] <-> Ch2 Sample 1/Ch2 Value
//     PlcTaskFast Inputs/GVL02_IO_EK1101.aOsInputFromEL4732Out1[2] <-> Ch2 Sample 2/Ch2 Value
//     PlcTaskFast Inputs/GVL02_IO_EK1101.aOsInputFromEL4732Out1[3] <-> Ch2 Sample 3/Ch2 Value
//     PlcTaskFast Inputs/GVL02_IO_EK1101.aOsInputFromEL4732Out1[4] <-> Ch2 Sample 4/Ch2 Value
//     PlcTaskFast Inputs/GVL02_IO_EK1101.aOsInputFromEL4732Out1[5] <-> Ch2 Sample 5/Ch2 Value
//     PlcTaskFast Inputs/GVL02_IO_EK1101.aOsInputFromEL4732Out1[6] <-> Ch2 Sample 6/Ch2 Value
//     PlcTaskFast Inputs/GVL02_IO_EK1101.aOsInputFromEL4732Out1[7] <-> Ch2 Sample 7/Ch2 Value
//     PlcTaskFast Inputs/GVL02_IO_EK1101.aOsInputFromEL4732Out1[8] <-> Ch2 Sample 8/Ch2 Value
//     PlcTaskFast Inputs/GVL02_IO_EK1101.aOsInputFromEL4732Out1[9] <-> Ch2 Sample 9/Ch2 Value
//   PLC1/PLC1 Instance <-> Device 1 (EtherCAT)/Term 21 (EK1101)/Term 27 (EL4732)
//     PlcTask Outputs/GVL02_IO_EK1101.aOsOutputToEL3702In2[0] <-> Ch1 Sample 0/Ch1 Value
//     PlcTask Outputs/GVL02_IO_EK1101.aOsOutputToEL3702In2[10] <-> Ch1 Sample 10/Ch1 Value
//     PlcTask Outputs/GVL02_IO_EK1101.aOsOutputToEL3702In2[11] <-> Ch1 Sample 11/Ch1 Value
//     PlcTask Outputs/GVL02_IO_EK1101.aOsOutputToEL3702In2[12] <-> Ch1 Sample 12/Ch1 Value
//     PlcTask Outputs/GVL02_IO_EK1101.aOsOutputToEL3702In2[13] <-> Ch1 Sample 13/Ch1 Value
//     PlcTask Outputs/GVL02_IO_EK1101.aOsOutputToEL3702In2[14] <-> Ch1 Sample 14/Ch1 Value
//     PlcTask Outputs/GVL02_IO_EK1101.aOsOutputToEL3702In2[15] <-> Ch1 Sample 15/Ch1 Value
//     PlcTask Outputs/GVL02_IO_EK1101.aOsOutputToEL3702In2[16] <-> Ch1 Sample 16/Ch1 Value
//     PlcTask Outputs/GVL02_IO_EK1101.aOsOutputToEL3702In2[17] <-> Ch1 Sample 17/Ch1 Value
//     PlcTask Outputs/GVL02_IO_EK1101.aOsOutputToEL3702In2[18] <-> Ch1 Sample 18/Ch1 Value
//     PlcTask Outputs/GVL02_IO_EK1101.aOsOutputToEL3702In2[19] <-> Ch1 Sample 19/Ch1 Value
//     PlcTask Outputs/GVL02_IO_EK1101.aOsOutputToEL3702In2[1] <-> Ch1 Sample 1/Ch1 Value
//     PlcTask Outputs/GVL02_IO_EK1101.aOsOutputToEL3702In2[20] <-> Ch1 Sample 20/Ch1 Value
//     PlcTask Outputs/GVL02_IO_EK1101.aOsOutputToEL3702In2[21] <-> Ch1 Sample 21/Ch1 Value
//     PlcTask Outputs/GVL02_IO_EK1101.aOsOutputToEL3702In2[22] <-> Ch1 Sample 22/Ch1 Value
//     PlcTask Outputs/GVL02_IO_EK1101.aOsOutputToEL3702In2[23] <-> Ch1 Sample 23/Ch1 Value
//     PlcTask Outputs/GVL02_IO_EK1101.aOsOutputToEL3702In2[24] <-> Ch1 Sample 24/Ch1 Value
//     PlcTask Outputs/GVL02_IO_EK1101.aOsOutputToEL3702In2[25] <-> Ch1 Sample 25/Ch1 Value
//     PlcTask Outputs/GVL02_IO_EK1101.aOsOutputToEL3702In2[26] <-> Ch1 Sample 26/Ch1 Value
//     PlcTask Outputs/GVL02_IO_EK1101.aOsOutputToEL3702In2[27] <-> Ch1 Sample 27/Ch1 Value
//     PlcTask Outputs/GVL02_IO_EK1101.aOsOutputToEL3702In2[28] <-> Ch1 Sample 28/Ch1 Value
//     PlcTask Outputs/GVL02_IO_EK1101.aOsOutputToEL3702In2[29] <-> Ch1 Sample 29/Ch1 Value
//     PlcTask Outputs/GVL02_IO_EK1101.aOsOutputToEL3702In2[2] <-> Ch1 Sample 2/Ch1 Value
//     PlcTask Outputs/GVL02_IO_EK1101.aOsOutputToEL3702In2[30] <-> Ch1 Sample 30/Ch1 Value
//     PlcTask Outputs/GVL02_IO_EK1101.aOsOutputToEL3702In2[31] <-> Ch1 Sample 31/Ch1 Value
//     PlcTask Outputs/GVL02_IO_EK1101.aOsOutputToEL3702In2[32] <-> Ch1 Sample 32/Ch1 Value
//     PlcTask Outputs/GVL02_IO_EK1101.aOsOutputToEL3702In2[33] <-> Ch1 Sample 33/Ch1 Value
//     PlcTask Outputs/GVL02_IO_EK1101.aOsOutputToEL3702In2[34] <-> Ch1 Sample 34/Ch1 Value
//     PlcTask Outputs/GVL02_IO_EK1101.aOsOutputToEL3702In2[35] <-> Ch1 Sample 35/Ch1 Value
//     PlcTask Outputs/GVL02_IO_EK1101.aOsOutputToEL3702In2[36] <-> Ch1 Sample 36/Ch1 Value
//     PlcTask Outputs/GVL02_IO_EK1101.aOsOutputToEL3702In2[37] <-> Ch1 Sample 37/Ch1 Value
//     PlcTask Outputs/GVL02_IO_EK1101.aOsOutputToEL3702In2[38] <-> Ch1 Sample 38/Ch1 Value
//     PlcTask Outputs/GVL02_IO_EK1101.aOsOutputToEL3702In2[39] <-> Ch1 Sample 39/Ch1 Value
//     PlcTask Outputs/GVL02_IO_EK1101.aOsOutputToEL3702In2[3] <-> Ch1 Sample 3/Ch1 Value
//     PlcTask Outputs/GVL02_IO_EK1101.aOsOutputToEL3702In2[40] <-> Ch1 Sample 40/Ch1 Value
//     PlcTask Outputs/GVL02_IO_EK1101.aOsOutputToEL3702In2[41] <-> Ch1 Sample 41/Ch1 Value
//     PlcTask Outputs/GVL02_IO_EK1101.aOsOutputToEL3702In2[42] <-> Ch1 Sample 42/Ch1 Value
//     PlcTask Outputs/GVL02_IO_EK1101.aOsOutputToEL3702In2[43] <-> Ch1 Sample 43/Ch1 Value
//     PlcTask Outputs/GVL02_IO_EK1101.aOsOutputToEL3702In2[44] <-> Ch1 Sample 44/Ch1 Value
//     PlcTask Outputs/GVL02_IO_EK1101.aOsOutputToEL3702In2[45] <-> Ch1 Sample 45/Ch1 Value
//     PlcTask Outputs/GVL02_IO_EK1101.aOsOutputToEL3702In2[46] <-> Ch1 Sample 46/Ch1 Value
//     PlcTask Outputs/GVL02_IO_EK1101.aOsOutputToEL3702In2[47] <-> Ch1 Sample 47/Ch1 Value
//     PlcTask Outputs/GVL02_IO_EK1101.aOsOutputToEL3702In2[48] <-> Ch1 Sample 48/Ch1 Value
//     PlcTask Outputs/GVL02_IO_EK1101.aOsOutputToEL3702In2[49] <-> Ch1 Sample 49/Ch1 Value
//     PlcTask Outputs/GVL02_IO_EK1101.aOsOutputToEL3702In2[4] <-> Ch1 Sample 4/Ch1 Value
//     PlcTask Outputs/GVL02_IO_EK1101.aOsOutputToEL3702In2[50] <-> Ch1 Sample 50/Ch1 Value
//     PlcTask Outputs/GVL02_IO_EK1101.aOsOutputToEL3702In2[51] <-> Ch1 Sample 51/Ch1 Value
//     PlcTask Outputs/GVL02_IO_EK1101.aOsOutputToEL3702In2[52] <-> Ch1 Sample 52/Ch1 Value
//     PlcTask Outputs/GVL02_IO_EK1101.aOsOutputToEL3702In2[53] <-> Ch1 Sample 53/Ch1 Value
//     PlcTask Outputs/GVL02_IO_EK1101.aOsOutputToEL3702In2[54] <-> Ch1 Sample 54/Ch1 Value
//     PlcTask Outputs/GVL02_IO_EK1101.aOsOutputToEL3702In2[55] <-> Ch1 Sample 55/Ch1 Value
//     PlcTask Outputs/GVL02_IO_EK1101.aOsOutputToEL3702In2[56] <-> Ch1 Sample 56/Ch1 Value
//     PlcTask Outputs/GVL02_IO_EK1101.aOsOutputToEL3702In2[57] <-> Ch1 Sample 57/Ch1 Value
//     PlcTask Outputs/GVL02_IO_EK1101.aOsOutputToEL3702In2[58] <-> Ch1 Sample 58/Ch1 Value
//     PlcTask Outputs/GVL02_IO_EK1101.aOsOutputToEL3702In2[59] <-> Ch1 Sample 59/Ch1 Value
//     PlcTask Outputs/GVL02_IO_EK1101.aOsOutputToEL3702In2[5] <-> Ch1 Sample 5/Ch1 Value
//     PlcTask Outputs/GVL02_IO_EK1101.aOsOutputToEL3702In2[60] <-> Ch1 Sample 60/Ch1 Value
//     PlcTask Outputs/GVL02_IO_EK1101.aOsOutputToEL3702In2[61] <-> Ch1 Sample 61/Ch1 Value
//     PlcTask Outputs/GVL02_IO_EK1101.aOsOutputToEL3702In2[62] <-> Ch1 Sample 62/Ch1 Value
//     PlcTask Outputs/GVL02_IO_EK1101.aOsOutputToEL3702In2[63] <-> Ch1 Sample 63/Ch1 Value
//     PlcTask Outputs/GVL02_IO_EK1101.aOsOutputToEL3702In2[64] <-> Ch1 Sample 64/Ch1 Value
//     PlcTask Outputs/GVL02_IO_EK1101.aOsOutputToEL3702In2[65] <-> Ch1 Sample 65/Ch1 Value
//     PlcTask Outputs/GVL02_IO_EK1101.aOsOutputToEL3702In2[66] <-> Ch1 Sample 66/Ch1 Value
//     PlcTask Outputs/GVL02_IO_EK1101.aOsOutputToEL3702In2[67] <-> Ch1 Sample 67/Ch1 Value
//     PlcTask Outputs/GVL02_IO_EK1101.aOsOutputToEL3702In2[68] <-> Ch1 Sample 68/Ch1 Value
//     PlcTask Outputs/GVL02_IO_EK1101.aOsOutputToEL3702In2[69] <-> Ch1 Sample 69/Ch1 Value
//     PlcTask Outputs/GVL02_IO_EK1101.aOsOutputToEL3702In2[6] <-> Ch1 Sample 6/Ch1 Value
//     PlcTask Outputs/GVL02_IO_EK1101.aOsOutputToEL3702In2[70] <-> Ch1 Sample 70/Ch1 Value
//     PlcTask Outputs/GVL02_IO_EK1101.aOsOutputToEL3702In2[71] <-> Ch1 Sample 71/Ch1 Value
//     PlcTask Outputs/GVL02_IO_EK1101.aOsOutputToEL3702In2[72] <-> Ch1 Sample 72/Ch1 Value
//     PlcTask Outputs/GVL02_IO_EK1101.aOsOutputToEL3702In2[73] <-> Ch1 Sample 73/Ch1 Value
//     PlcTask Outputs/GVL02_IO_EK1101.aOsOutputToEL3702In2[74] <-> Ch1 Sample 74/Ch1 Value
//     PlcTask Outputs/GVL02_IO_EK1101.aOsOutputToEL3702In2[75] <-> Ch1 Sample 75/Ch1 Value
//     PlcTask Outputs/GVL02_IO_EK1101.aOsOutputToEL3702In2[76] <-> Ch1 Sample 76/Ch1 Value
//     PlcTask Outputs/GVL02_IO_EK1101.aOsOutputToEL3702In2[77] <-> Ch1 Sample 77/Ch1 Value
//     PlcTask Outputs/GVL02_IO_EK1101.aOsOutputToEL3702In2[78] <-> Ch1 Sample 78/Ch1 Value
//     PlcTask Outputs/GVL02_IO_EK1101.aOsOutputToEL3702In2[79] <-> Ch1 Sample 79/Ch1 Value
//     PlcTask Outputs/GVL02_IO_EK1101.aOsOutputToEL3702In2[7] <-> Ch1 Sample 7/Ch1 Value
//     PlcTask Outputs/GVL02_IO_EK1101.aOsOutputToEL3702In2[80] <-> Ch1 Sample 80/Ch1 Value
//     PlcTask Outputs/GVL02_IO_EK1101.aOsOutputToEL3702In2[81] <-> Ch1 Sample 81/Ch1 Value
//     PlcTask Outputs/GVL02_IO_EK1101.aOsOutputToEL3702In2[82] <-> Ch1 Sample 82/Ch1 Value
//     PlcTask Outputs/GVL02_IO_EK1101.aOsOutputToEL3702In2[83] <-> Ch1 Sample 83/Ch1 Value
//     PlcTask Outputs/GVL02_IO_EK1101.aOsOutputToEL3702In2[84] <-> Ch1 Sample 84/Ch1 Value
//     PlcTask Outputs/GVL02_IO_EK1101.aOsOutputToEL3702In2[85] <-> Ch1 Sample 85/Ch1 Value
//     PlcTask Outputs/GVL02_IO_EK1101.aOsOutputToEL3702In2[86] <-> Ch1 Sample 86/Ch1 Value
//     PlcTask Outputs/GVL02_IO_EK1101.aOsOutputToEL3702In2[87] <-> Ch1 Sample 87/Ch1 Value
//     PlcTask Outputs/GVL02_IO_EK1101.aOsOutputToEL3702In2[88] <-> Ch1 Sample 88/Ch1 Value
//     PlcTask Outputs/GVL02_IO_EK1101.aOsOutputToEL3702In2[89] <-> Ch1 Sample 89/Ch1 Value
//     PlcTask Outputs/GVL02_IO_EK1101.aOsOutputToEL3702In2[8] <-> Ch1 Sample 8/Ch1 Value
//     PlcTask Outputs/GVL02_IO_EK1101.aOsOutputToEL3702In2[90] <-> Ch1 Sample 90/Ch1 Value
//     PlcTask Outputs/GVL02_IO_EK1101.aOsOutputToEL3702In2[91] <-> Ch1 Sample 91/Ch1 Value
//     PlcTask Outputs/GVL02_IO_EK1101.aOsOutputToEL3702In2[92] <-> Ch1 Sample 92/Ch1 Value
//     PlcTask Outputs/GVL02_IO_EK1101.aOsOutputToEL3702In2[93] <-> Ch1 Sample 93/Ch1 Value
//     PlcTask Outputs/GVL02_IO_EK1101.aOsOutputToEL3702In2[94] <-> Ch1 Sample 94/Ch1 Value
//     PlcTask Outputs/GVL02_IO_EK1101.aOsOutputToEL3702In2[95] <-> Ch1 Sample 95/Ch1 Value
//     PlcTask Outputs/GVL02_IO_EK1101.aOsOutputToEL3702In2[96] <-> Ch1 Sample 96/Ch1 Value
//     PlcTask Outputs/GVL02_IO_EK1101.aOsOutputToEL3702In2[97] <-> Ch1 Sample 97/Ch1 Value
//     PlcTask Outputs/GVL02_IO_EK1101.aOsOutputToEL3702In2[98] <-> Ch1 Sample 98/Ch1 Value
//     PlcTask Outputs/GVL02_IO_EK1101.aOsOutputToEL3702In2[99] <-> Ch1 Sample 99/Ch1 Value
//     PlcTask Outputs/GVL02_IO_EK1101.aOsOutputToEL3702In2[9] <-> Ch1 Sample 9/Ch1 Value
//     PlcTask Outputs/GVL02_IO_EK1101.nEL4732Ch1CycleCount <-> Ch1 CycleCount/Ch1 CycleCount
//   PLC1/PLC1 Instance <-> MC3 Project/Axes/LoadControl (FluidPower Axis)
//     FluidPowerSim Inputs/LoadControlSim.SetVelo <-> Analog Outputs/Output
//     FluidPowerSim Outputs/LoadControlSim.ActPos <-> SSI Inputs/Counter Value
//     PlcTask Inputs/LoadControl.HydAxis.McToPlc/Act <-> McToPlc/Act
//     PlcTask Inputs/LoadControl.HydAxis.McToPlc/FluidPower <-> McToPlc/FluidPower
//     PlcTask Inputs/LoadControl.HydAxis.McToPlc/LoadControl <-> McToPlc/LoadControl
//     PlcTask Inputs/LoadControl.HydAxis.McToPlc/Set <-> McToPlc/Set
//     PlcTask Inputs/LoadControl.HydAxis.McToPlc/Std <-> McToPlc/Std
//     PlcTask Outputs/LoadControl.HydAxis.PlcToMc/Std <-> PlcToMc/Std
//   PLC1/PLC1 Instance <-> MC3 Project/Axes/LoadControl (FluidPower Axis)/Pressure Sensor A
//     FluidPowerSim Outputs/LoadControlSim.PressureA <-> Analog Inputs/Counter Value
//   PLC1/PLC1 Instance <-> MC3 Project/Axes/Master (Axis)
//     PlcTask Inputs/MC3_Gearing.Axis[0].McToPlc/Act <-> McToPlc/Act
//     PlcTask Inputs/MC3_Gearing.Axis[0].McToPlc/Set <-> McToPlc/Set
//     PlcTask Inputs/MC3_Gearing.Axis[0].McToPlc/Std <-> McToPlc/Std
//     PlcTask Outputs/MC3_Gearing.Axis[0].PlcToMc/Std <-> PlcToMc/Std
//   PLC1/PLC1 Instance <-> MC3 Project/Axes/Nc2_Slave (Axis)
//     PlcTask Inputs/ExtSetpoint_MC3_NC2.Mc3SlaveAxis.McToPlc/Act <-> McToPlc/Act
//     PlcTask Inputs/ExtSetpoint_MC3_NC2.Mc3SlaveAxis.McToPlc/Set <-> McToPlc/Set
//     PlcTask Inputs/ExtSetpoint_MC3_NC2.Mc3SlaveAxis.McToPlc/Std <-> McToPlc/Std
//     PlcTask Outputs/ExtSetpoint_MC3_NC2.Mc3SlaveAxis.PlcToMc/Std <-> PlcToMc/Std
//   PLC1/PLC1 Instance <-> MC3 Project/Axes/PressToTarget (FluidPower Axis)
//     FluidPowerSim Inputs/PressToTargetSim.SetVelo <-> Analog Outputs/Output
//     FluidPowerSim Outputs/PressToTargetSim.ActPos <-> SSI Inputs/Counter Value
//     PlcTask Inputs/PressToTarget.HydAxis.McToPlc/Act <-> McToPlc/Act
//     PlcTask Inputs/PressToTarget.HydAxis.McToPlc/FluidPower <-> McToPlc/FluidPower
//     PlcTask Inputs/PressToTarget.HydAxis.McToPlc/LoadControl <-> McToPlc/LoadControl
//     PlcTask Inputs/PressToTarget.HydAxis.McToPlc/Set <-> McToPlc/Set
//     PlcTask Inputs/PressToTarget.HydAxis.McToPlc/Std <-> McToPlc/Std
//     PlcTask Outputs/PressToTarget.HydAxis.PlcToMc/Std <-> PlcToMc/Std
//   PLC1/PLC1 Instance <-> MC3 Project/Axes/PressToTarget (FluidPower Axis)/Pressure Sensor A
//     FluidPowerSim Outputs/PressToTargetSim.PressureA <-> Analog Inputs/Counter Value
//   PLC1/PLC1 Instance <-> MC3 Project/Axes/Reversing (Axis)
//     PlcTask Inputs/MC3_ReversingSequence.ax1.McToPlc/Act <-> McToPlc/Act
//     PlcTask Inputs/MC3_ReversingSequence.ax1.McToPlc/Set <-> McToPlc/Set
//     PlcTask Inputs/MC3_ReversingSequence.ax1.McToPlc/Std <-> McToPlc/Std
//     PlcTask Outputs/MC3_ReversingSequence.ax1.PlcToMc/Std <-> PlcToMc/Std
//   PLC1/PLC1 Instance <-> MC3 Project/Axes/Slave (Axis)
//     PlcTask Inputs/MC3_Gearing.Axis[1].McToPlc/Act <-> McToPlc/Act
//     PlcTask Inputs/MC3_Gearing.Axis[1].McToPlc/Set <-> McToPlc/Set
//     PlcTask Inputs/MC3_Gearing.Axis[1].McToPlc/Std <-> McToPlc/Std
//     PlcTask Outputs/MC3_Gearing.Axis[1].PlcToMc/Std <-> PlcToMc/Std
//   PLC1/PLC1 Instance <-> NC-Task 1 SAF/Axes/Axis 1 Stepper
//     PlcTask Inputs/GVL20_Axis.stAxis1.NcToPlc <-> Outputs/ToPlc
//     PlcTask Outputs/GVL20_Axis.stAxis1.PlcToNc <-> Inputs/FromPlc
//   PLC1/PLC1 Instance <-> NC-Task 1 SAF/Axes/Axis 2 Servo EL
//     PlcTask Inputs/GVL20_Axis.stAxis2.NcToPlc <-> Outputs/ToPlc
//     PlcTask Outputs/GVL20_Axis.stAxis2.PlcToNc <-> Inputs/FromPlc
//   PLC1/PLC1 Instance <-> NC-Task 1 SAF/Axes/Axis 3 Servo A AX
//     PlcTask Inputs/GVL20_Axis.stAxis3.NcToPlc <-> Outputs/ToPlc
//     PlcTask Outputs/GVL20_Axis.stAxis3.PlcToNc <-> Inputs/FromPlc
//   PLC1/PLC1 Instance <-> NC-Task 1 SAF/Axes/Axis 4 Servo B AX
//     PlcTask Inputs/GVL20_Axis.stAxis4.NcToPlc <-> Outputs/ToPlc
//     PlcTask Outputs/GVL20_Axis.stAxis4.PlcToNc <-> Inputs/FromPlc
//   PLC1/PLC1 Instance <-> NC-Task 1 SAF/Axes/Axis 5 Handwheel
//     PlcTask Inputs/GVL20_Axis.stAxis5.NcToPlc <-> Outputs/ToPlc
//     PlcTask Outputs/GVL20_Axis.stAxis5.PlcToNc <-> Inputs/FromPlc
//   PLC1/PLC1 Instance <-> NC-Task 1 SAF/Axes/MC3_ExtMaster
//     NC_Task_1_SAF Inputs/GVL.Nc2MasterAxis.NcToPlc <-> Outputs/ToPlc
//     NC_Task_1_SAF Outputs/GVL.Nc2MasterAxis.PlcToNc <-> Inputs/FromPlc
//   PLC1/PLC1 Instance <-> NC-Task 1 SAF/NCI
//     PlcTask Inputs/NCI.in_stItpToPlc <-> Outputs/ToPlc
//     PlcTask Outputs/NCI.out_stPlcToItp <-> Inputs/FromPlc

CONFIGURATION PLC1
    RESOURCE PLC ON TwinCAT3
        TASK FluidPowerSim(INTERVAL := T#2ms, PRIORITY := 16);
        TASK NC_Task_1_SAF(INTERVAL := T#1ms, PRIORITY := 6);
        TASK PlcTask(INTERVAL := T#1ms, PRIORITY := 8);
        PROGRAM PressToTargetSim WITH FluidPowerSim : PressToTargetSim;
        PROGRAM LoadControlSim WITH FluidPowerSim : LoadControlSim;
        PROGRAM PRG_SAF WITH NC_Task_1_SAF : PRG_SAF;
        PROGRAM MAIN WITH PlcTask : MAIN;
    END_RESOURCE
END_CONFIGURATION

// ---- POUs/MC3/ExternalSetpoint_Mc3_Nc2/Support/E_Command.TcDUT
TYPE E_Command :
(
    none := 0,
    Start,
    Stop,
	MoveSlaveVelo,
    Reset
);
END_TYPE

// ---- POUs/MC3/ExternalSetpoint_Mc3_Nc2/Support/E_State.TcDUT
TYPE E_State :
(
    Init := 0,
    Idle,
	ActivateExtSg,
    Run,
    StoppingSlave,
	StoppingMaster,
    Error,
    Resetting 
);
END_TYPE

// ---- POUs/MC3/Gearing/Support/E_Axis.TcDUT
{attribute 'to_string'}
TYPE E_Axis : (
		Master := 0,
		Slave
	);
END_TYPE

// ---- POUs/MC3/Gearing/Support/E_GearCommand.TcDUT
{attribute 'qualified_only'}
{attribute 'strict'}
{attribute 'to_string'}
TYPE E_GearCommand : (
		Idle := 0,
		Enable,
		Disable,
		GearInStationary,
		GearInVelocity,
		GearInPosition
	);
END_TYPE

// ---- GVLs/GVL.TcGVL
VAR_GLOBAL CONSTANT
	iMAX_AXES_REF : INT := 5;
END_VAR

VAR_GLOBAL
	iGlobalCounter : UINT;
	fbCrititcalSection : FB_IecCriticalSection;
END_VAR

VAR_GLOBAL
	{attribute 'TcContextName':='NC SAF'}
	Nc2MasterAxis : Tc2_MC2.AXIS_REF;
END_VAR

// ---- GVLs/GVL20_Axis.TcGVL
(* GVL20_Axis - Global variables axis *)
{attribute 'TcContextName' := 'PlcTask'}
VAR_GLOBAL
	
(* Axis 1 inputs and outputs *)
	stAxis1									:Tc2_Mc2.AXIS_REF;

(* Axis 2 inputs and outputs *)
	stAxis2									:Tc2_Mc2.AXIS_REF;

(* Axis 3 - 4 (AX5203) inputs and outputs *)
	nAxis3TorqueFeedback			AT%I*	:INT;		(* Axis 3 current +/- 1000 *)
	nAxis4TorqueFeedback			AT%I*	:INT;		(* Axis 4 current +/- 1000 *)

	nAX5203DigitalInputs			AT%I*	:UINT;		(* Digital inputs AX5000
															BIT 0 - servo reference cam (axis 3)
															BIT 1 - servo reference cam (axis 4)
															BIT 2 - switch S26
															BIT 3 - switch S27 *)

	nAX5203DigitalOutputs			AT%Q*	:UINT;		(* Digital output AX5000 
															BIT 7 - Led H27 *)
	
	stAxis3									:Tc2_Mc2.AXIS_REF;
	stAxis4									:Tc2_Mc2.AXIS_REF;

(* Axis 5 (Handwheel) inputs and outputs *)
	stAxis5									:Tc2_Mc2.AXIS_REF;

END_VAR
(* End *)

// ---- POUs/MC3/PressToTarget/PressToTargetSim.TcPOU
PROGRAM PressToTargetSim
VAR
	ActPos AT%Q*:	DINT;
	SetVelo AT%I*:	INT;
	PressureA AT%Q*:	INT;
 
 	fSetVelo:	LREAL;
 	fActPos:	LREAL;
	fPressureA:	LREAL;

	bBrake: BOOL;
END_VAR



fSetVelo:=INT_TO_LREAL(SetVelo)/32767*500.0;

fActPos:=fActPos+fSetVelo*0.002;

fActPos:=MIN(MAX(fActPos,0.0),200.0);
ActPos:=LREAL_TO_DINT(fActPos * 1000.0);

fPressureA:=MIN(MAX((fActPos-100.0)*5,0.0),200.0); 

IF bBrake THEN
	fPressureA:=MIN(MAX((fActPos-100.0)*5,0.0),20.0); 
END_IF
PressureA:=LREAL_TO_INT(fPressureA/400.0*32767);

END_PROGRAM

// ---- POUs/MC3/LoadControl/LoadControlSim.TcPOU
PROGRAM LoadControlSim
VAR
	ActPos AT%Q*:	DINT;
	SetVelo AT%I*:	INT;
	PressureA AT%Q*:	INT;
 
 	fSetVelo:	LREAL;
 	fActPos:	LREAL;
	fPressureA:	LREAL;

	bBrake: BOOL;
END_VAR



fSetVelo:=INT_TO_LREAL(SetVelo)/32767*500.0;

fActPos:=fActPos+fSetVelo*0.001;

fActPos:=MIN(MAX(fActPos,0.0),500.0);
ActPos:=LREAL_TO_DINT(fActPos * 1000.0);

fPressureA:=MIN(MAX((fActPos-100.0)*5,0.0),200.0); 

IF bBrake THEN
	fPressureA:=MIN(MAX((fActPos-100.0)*5,0.0),20.0); 
END_IF
PressureA:=LREAL_TO_INT(fPressureA/400.0*32767);

END_PROGRAM

// ---- POUs/MC3/ExternalSetpoint_Mc3_Nc2/PRG_SAF.TcPOU
PROGRAM PRG_SAF
VAR
END_VAR

Nc2MasterAxis();

END_PROGRAM

// ---- POUs/MainPOUs/MAIN.TcPOU
PROGRAM MAIN
(*******************************************************************************************************
Title				:	Main program 
Description			:	Calling the created subroutines (Task 1ms)
Version / Date		:	1.0.0 / 23.05.2016 / created program (Version progress see below)

Supported hardware	: 	Demo-Rack (LAGE version)

Used Documentation	:	
Documentation	
Version/Date 		:	

Required libraries 	: 	Please look in the "References" folder
********************************************************************************************************)
VAR
	
(* Cycle counter *)
	nCycleCounter							:UDINT;

(* act_SUps - 1s UPS - Uninterruptible power supply *)
	fbSUps									:FB_S_UPS_CX51x0 := (eUpsMode:=eSUPS_WrPersistData_Shutdown);
	bPowerFailDetect						:BOOL;

(* act_SystemStart *)
	eStateSystemStartSeq					:E_SystemStartupSequence;
	eSystemStartSeqErrStep					:E_SystemStartupSequence := eSystemStart_NoError;
	bSystemStartErr							:BOOL;
	bSystemStartEnd							:BOOL;
	fbTimerSystemStart						:TON;


(*******************************************************************************************************
Version / Date / Description:
1.0.0   / 23.05.2016 / created program
********************************************************************************************************)
(* End *)

	{attribute 'TcContextName':='PlcTask'}
	iCounter AT %Q*		: DINT;
	
	//fbMC2				: FB_MC2;
	//fbNCI				: FB_NCI;
	fbOOPAxisTable		: FB_OOPAxisTable;
	fbOOPCylReg			: FB_OOPCylinderRegulator;
	fbOOPConveyor		: FB_OOPConveyor;
	
	{attribute 'TcAnalytics'}
	fbScope				: FB_GenerateData;
	fbUmlSc				: FB_UML_SC_Composite;
	fbUmlSc_Lamp		: FB_UML_SC_Lamp;

	fbModeChangeTimer	: TON := (PT := T#60S);
	nRemainingModeTime	: UDINT;
	
	eSampleMode			: E_SampleMode;	
	eSampleModeMC2		: E_SampleMode;	
	eSampleModeNCI		: E_SampleMode;	
	eSampleModeOOP		: E_SampleMode;	
	eSampleModeOOPConv	: E_SampleMode;	

	nRadioButton		: INT;
	AxisRef				: ARRAY [1..iMAX_AXES_REF] OF Tc2_Mc2.AXIS_REF;			// axis reference (process data plc/nc)
	
	{attribute 'TcContextName':='PlcTask'}
	wFrmXWcState_MAIN AT %I*	: WORD; 			// link to NC-task related ethercat frame state (Frm0WcState)
	x1: WORD;
	
	fblog : FB_RTMon_LogMark;

END_VAR

(* MAIN - 1ms *)

(* THIS CODE IS ONLY AN EXAMPLE - YOU HAVE TO CHECK APTITUDE FOR YOUR APPLICATION *)

(* Cycle counter *)
	nCycleCounter := nCycleCounter + 1;


(* 1s USV *)
	act_SUps();


(* Startup detect *)
	IF TwinCAT_SystemInfoVarList._TaskInfo[GETCURTASKINDEXEX()].FirstCycle
	THEN
		bFirstCycleDetected	:= TRUE;
	END_IF


(* Startup- or machine sequence *)
	IF bFirstCycleDetected
	THEN
	(* Startup sequenz *)
		act_SystemStart();

		IF bSystemStartEnd
		THEN
			bFirstCycleDetected := FALSE;
			bMachineSequenzAktiv := TRUE;
		END_IF

	ELSIF bMachineSequenzAktiv
	THEN
	(* Machine sequenz *)
		(* Test general *)
			GeneralPlc();
		
		(* Test blinker *)
			Blinker();

		(* Test clock generator *)
			ClockGenerator();
		
		(* Test axis *)
			AxisGeneral();
			Axis1();
			Axis2();
			Axis3();
			Axis4();
			stAxis5.ReadStatus();

		(* Test EtherCAT diacnostic *)
			DiagnosticEtherCAT();
			
		(* Test - XFC - extrem fast control *)	
			DcTimes();
			AnalogOutputOversampling();
			PositionCamTimeStampAxis2();
			SignalLengthMeasurementCamAxis2();
			TouchProbeTimeStampCamAxis2();

		(* Test TwinSAFE *)	
			TwinSAFE();
		
	END_IF

(* End *)

iCounter := iCounter + 1;

//switch mode (MC2, NCI, OOP)
A_ModeSwitch();

(*//call MC2 sample
fblog.LogStart(1,0); //added this
fbMC2(AxisRef := AxisRef, eSampleModeIn := eSampleMode, eSampleModeOut => eSampleModeMC2);
fblog.LogStop(1,0); // added this*)


//call NCI sample
fblog.LogStart(2,0); //added this
NCI();
//fbNCI(AxisRef := AxisRef, eSampleModeIn := eSampleMode, eSampleModeOut => eSampleModeNCI);
fblog.LogStop(2,0);

//Call Cam Table Sample
CamTable();

//Call External Setpoint Generator Sample
Ext_SP_Gen();

//call OOP sample
fblog.LogStart(3,0);
fbOOPAxisTable(AxisRef := AxisRef, eSampleModeIn := eSampleMode, eSampleModeOut => eSampleModeOOP);
fbOOPCylReg();
fblog.LogStop(3,0);

//call OOP conveyor sample
fblog.logstart(4,0);
fbOOPConveyor(AxisRef := AxisRef, eSampleModeIn := eSampleMode, eSampleModeOut => eSampleModeOOPConv);
fblog.logstop(4,0);

//call language samples
fblog.LogMark(5,0);
MAIN_CFC();					//continuous flow chart
fblog.LogMark(5,1);
MAIN_CFC_PageOriented();	//continuous flow chart, page oriented
fblog.LogMark(5,2);
MAIN_FBD_IL_LD();			//use language switching via menu "FBD/IL/LD, function block diagram, instruction list, ladder logic 
fblog.LogMark(5,3);
MAIN_SFC();					//sequential flow chart 
fblog.LogMark(5,4);
MAIN_ST();					//structured text
fblog.LogStop(5,0);


//call UML SC composite sample
fblog.LogStart(6,0);
fbUmlSc();
fbUmlSc_Lamp();
fblog.LogStop(6,0);

x1 := wFrmXWcState_MAIN;

//Call TwinSAFE Program
TwinSAFE();

//Call IoT Program
IoT_JSON_XML();

//Call Database Server Sample
CSVSample();

//Call MC3 Samples
MC3_ReversingSequence();
ExtSetpoint_MC3_NC2();
MC3_Gearing();
PressToTarget();
LoadControl();

ACTION A_ModeSwitch:
//decide for an active motion sample
fbModeChangeTimer(IN := TRUE);
nRemainingModeTime := TIME_TO_UDINT(fbModeChangeTimer.PT-fbModeChangeTimer.ET)/1000;

IF fbModeChangeTimer.Q OR (eSampleMode = eSMode_Idle) OR (nRadioButton > 0) THEN
	//switch if ready 
	
	IF (eSampleModeMC2 = eSMode_Idle) AND (eSampleModeNCI = eSMode_Idle) AND (eSampleModeOOP = eSMode_Idle) AND (eSampleModeOOPConv = eSMode_Idle) THEN
		//ready to switch
		fbModeChangeTimer(IN := FALSE);
		
		CASE eSampleMode OF
		eSMode_Idle:
			CASE nRadioButton OF
			1:
				eSampleMode := eSMode_MC2_Req;
			2:			
				eSampleMode := eSMode_NCI_Req;
			3:			
				eSampleMode := eSMode_OOP_Req;
			4:			
				eSampleMode := eSMode_OOPConv_Req;
			ELSE //idle
				eSampleMode := eSMode_MC2_Req;
			END_CASE
			
		eSMode_MC2_Req:
			CASE nRadioButton OF
			1:
				eSampleMode := eSMode_MC2_Req;
			2:			
				eSampleMode := eSMode_NCI_Req;
			3:			
				eSampleMode := eSMode_OOP_Req;
			4:			
				eSampleMode := eSMode_OOPConv_Req;
			ELSE //idle
				eSampleMode := eSMode_NCI_Req;
			END_CASE
			
		eSMode_NCI_Req:
			CASE nRadioButton OF
			1:
				eSampleMode := eSMode_MC2_Req;
			2:			
				eSampleMode := eSMode_NCI_Req;
			3:			
				eSampleMode := eSMode_OOP_Req;
			4:			
				eSampleMode := eSMode_OOPConv_Req;
			ELSE //idle
				eSampleMode := eSMode_OOP_Req;
			END_CASE
			
		eSMode_OOP_Req:
			CASE nRadioButton OF
			1:
				eSampleMode := eSMode_MC2_Req;
			2:			
				eSampleMode := eSMode_NCI_Req;
			3:			
				eSampleMode := eSMode_OOP_Req;
			4:			
				eSampleMode := eSMode_OOPConv_Req;
			ELSE //idle
				eSampleMode := eSMode_MC2_Req;
			END_CASE
			
		eSMode_OOPConv_Req:
			CASE nRadioButton OF
			1:
				eSampleMode := eSMode_MC2_Req;
			2:			
				eSampleMode := eSMode_NCI_Req;
			3:			
				eSampleMode := eSMode_OOP_Req;
			4:			
				eSampleMode := eSMode_OOPConv_Req;
			ELSE //idle
				eSampleMode := eSMode_MC2_Req;
			END_CASE
			
		ELSE
			eSampleMode := eSMode_MC2_Req;
		END_CASE
		
		nRadioButton := 0;
	END_IF 
END_IF
END_ACTION

ACTION act_SUps:
(* Aktion - 1s UPS - Uninterruptible power supply *)

	fbSUps(); (* see instance declaration for initalisation of eUpsMode parameter *) 

	(*
	Default Values of FB_S_UPS_CX51x0-Inputs:
						sNetID 			:=	'' -> local netid
						iPLCPort 		:=	AMSPORT_R0_PLC_RTS1 -> 801 = 1st PLC Runtime 
						iUPSPort		:=	16#588 -> Port for reading Power State of UPS
						tTimeout 		:=	DEFAULT_ADS_TIMEOUT -> 5S
						eUpsMode 		:=	eSUPS_WrPersistData_Shutdown -> writing persistent data + shutdown
						ePersistentMode :=	SPDM_2PASS -> All data is from same plc cycle, cycletime exceeds possible. Plc stops with the shutdown, a few cycles after writing persistent data. 
						tRecoverTime 	:=	T#10s -> 10s power to recover from short power failure before eSUPS_PowerOK is reported (in mode eSUPS_WrPersistData_NoShutdown/eSUPS_CheckPowerStatus)

	eUpsMode =							in case of powerfailure:
	 	eSUPS_WrPersistData_Shutdown 	->	writing of persistent data + shutdown
	 	eSUPS_WrPersistData_NoShutdown 	->	writing of PERSISTENT data, no shutdown
	 	eSUPS_CheckPowerStatus 			->	reports powerfailure without ACTION (no writing, no shutdown) 
	 	eSUPS_ImmediateShutdown 		->	skips writing of data, immediate shutdown
	*)	

(* Power fail detected *)
	IF fbSUps.bPowerFailDetect
		AND NOT bPowerFailDetect
	THEN
	
		(* Count the power failures *)
		nPowerFailureCounter := nPowerFailureCounter + 1;
		bPowerFailDetect	 := TRUE;
	
	ELSE

		IF NOT fbSUps.bPowerFailDetect
		THEN
			bPowerFailDetect:=FALSE;
		END_IF

	END_IF

(* End *)
END_ACTION

ACTION act_SystemStart:
(* Aktion system start *)

	CASE eStateSystemStartSeq OF

	
		eSystemStart_Start			: 	(* Waiting for start *)
		
				eStateSystemStartSeq := eSystemStart_Init;

				
		eSystemStart_Init			:	(* Initialize *)

				fbTimerSystemStart(IN := FALSE);
				eStateSystemStartSeq := eSystemStart_LedOn;

				
		eSystemStart_LedOn			:	(* Sequence Leds on *)

				fbTimerSystemStart(	
					IN := TRUE,
					PT := T#2250MS);

				bLedH10	:=	fbTimerSystemStart.ET > T#250MS;
				bLedH20 :=  bLedH10;
				bLedH31 :=  bLedH10;
				bLedH11	:=	fbTimerSystemStart.ET > T#500MS;
				bLedH21 :=  bLedH11;
				bLedH32 :=  bLedH11;
				bLedH12	:=	fbTimerSystemStart.ET > T#750MS;
				bLedH22 :=  bLedH12;
				bLedH33 :=  bLedH12;
				bLedH13	:=	fbTimerSystemStart.ET > T#1000MS;
				bLedH23 :=  bLedH13;
				bLedH14	:=	fbTimerSystemStart.ET > T#1250MS;
				bLedH24 :=  bLedH14;
				bLedH15	:=	fbTimerSystemStart.ET > T#1500MS;
				bLedH25 :=  bLedH15;
				bLedH16	:=	fbTimerSystemStart.ET > T#1750MS;
				bLedH26 :=  bLedH16;
				bLedH17	:=	fbTimerSystemStart.ET > T#2000MS;
				nAX5203DigitalOutputs.7 :=  bLedH17;

				IF fbTimerSystemStart.Q
				THEN
					fbTimerSystemStart(IN := FALSE);
					eStateSystemStartSeq := eSystemStart_LedOff;
				ELSIF FALSE
				THEN
					(* If error then notice the step *)
					eSystemStartSeqErrStep := eStateSystemStartSeq;
					eStateSystemStartSeq   := eSystemStart_ErrorStep;
				END_IF

				
		eSystemStart_LedOff			:	(* Sequence Leds off *)

				fbTimerSystemStart(	
					IN := TRUE,
					PT := T#2250MS);

				bLedH10	:=	fbTimerSystemStart.ET < T#250MS;
				bLedH20 :=  bLedH10;
				bLedH31 :=  bLedH10;
				bLedH11	:=	fbTimerSystemStart.ET < T#500MS;
				bLedH21 :=  bLedH11;
				bLedH32 :=  bLedH11;
				bLedH12	:=	fbTimerSystemStart.ET < T#750MS;
				bLedH22 :=  bLedH12;
				bLedH33 :=  bLedH12;
				bLedH13	:=	fbTimerSystemStart.ET < T#1000MS;
				bLedH23 :=  bLedH13;
				bLedH14	:=	fbTimerSystemStart.ET < T#1250MS;
				bLedH24 :=  bLedH14;
				bLedH15	:=	fbTimerSystemStart.ET < T#1500MS;
				bLedH25 :=  bLedH15;
				bLedH16	:=	fbTimerSystemStart.ET < T#1750MS;
				bLedH26 :=  bLedH16;
				bLedH17	:=	fbTimerSystemStart.ET < T#2000MS;
				nAX5203DigitalOutputs.7 :=  bLedH17;
									
				IF fbTimerSystemStart.Q
				THEN
					eStateSystemStartSeq := eSystemStart_Done;
				ELSIF FALSE
				THEN
					(* If error then notice the step *)
					eSystemStartSeqErrStep := eStateSystemStartSeq;
					eStateSystemStartSeq   := eSystemStart_ErrorStep;
				END_IF

				
		eSystemStart_Done			:	(* System start done *)

				bSystemStartEnd := TRUE;

				
		eSystemStart_ErrorStep		:	(* Error on system start *)

				bSystemStartErr := TRUE;

				IF FALSE
				THEN
					bSystemStartErr        := FALSE;
					eSystemStartSeqErrStep := eSystemStart_NoError;
					eStateSystemStartSeq   := eSystemStart_Start;
				END_IF 

	ELSE
		
		(* If not a valid step is active, then put on start *)
		eSystemStartSeqErrStep := eSystemStart_NoError;
		eStateSystemStartSeq   := eSystemStart_Start;
	
	END_CASE

(* End *)
END_ACTION

END_PROGRAM

// ---- POUs/Sample OOP/FB_OOPAxisTable.TcPOU
FUNCTION_BLOCK FB_OOPAxisTable
VAR_INPUT
	eSampleModeIn	: E_SampleMode;	
END_VAR
VAR_IN_OUT
	AxisRef			: ARRAY [1..iMAX_AXES_REF] OF Tc2_MC2.AXIS_REF;			// axis reference (process data plc/nc)
END_VAR
VAR_OUTPUT
	eSampleModeOut	: E_SampleMode;	
END_VAR
VAR
	iCounter 			: DINT;
END_VAR	
VAR
	//instances of axes FBs (of type FB_NcAxes or derived from FB_NcAxis, like AX5000, Servo Termins, Stepper, DC, ...)
	fbAX5000Axis1	: FB_AX5000Axis;
	fbAX5000Axis2	: FB_AX5000Axis;
	fbNcAxis		: FB_NcAxis;
		
	//interface pointers
	ipAxisX			: IAxis;
	ipAxisY			: IAxis;
	ipAxisZ			: IAxis;

	//device
	fbTable			: FB_Table;
	bExecute		: BOOL;
	bBusy			: BOOL;
	
	Timer			: TON := (PT := T#3s);
END_VAR

iCounter := iCounter + 1;

IF (eSampleModeIn = eSMode_OOP_Req) OR (eSampleModeOut = eSMode_OOP_Act) THEN
	//assign axes instances to the interface pointers
	ipAxisX := fbAX5000Axis1;
	ipAxisY := fbAX5000Axis2;
	ipAxisZ	:= fbNcAxis;
	
	//call axes with their axes references
	fbAX5000Axis1(sAxis	:= AxisRef[1]);
	fbAX5000Axis2(sAxis	:= AxisRef[2]);
	fbNcAxis(sAxis	:= AxisRef[3]);
	
	Timer(IN := TRUE);
	IF Timer.Q THEN
		Timer(IN := FALSE);
		bExecute := TRUE;
	END_IF
	
	//call device that uses axes via interface, therefore the axis type does not matter anymore
	fbTable(
		fbServoAxisX := ipAxisX,
		fbServoAxisY := ipAxisY,
		fbServoAxisZ := ipAxisZ,
		bExecute	 := bExecute,
		bBusy		 => bBusy
	);
		
	bExecute := FALSE;

	IF bBusy THEN
		eSampleModeOut := eSMode_OOP_Act;
	ELSE
		eSampleModeOut := eSMode_Idle;
	END_IF
END_IF

END_FUNCTION_BLOCK

// ---- POUs/Sample OOP/Table/Axis/FB_NcAxis.TcPOU
FUNCTION_BLOCK FB_NcAxis IMPLEMENTS IAxis
VAR_IN_OUT
	sAxis		: Tc2_Mc2.AXIS_REF;
END_VAR
VAR_INPUT
END_VAR
VAR_OUTPUT
	bActive		: BOOL;
	bBusy		: BOOL;
	bDone		: BOOL;
	bError		: BOOL;
	iErrorId	: UDINT;
	eCurState	: E_AxisState;
END_VAR
VAR
	//PLCopen FBs for axes
	fbMcPower	: Tc2_Mc2.MC_Power;
	fbMcReset	: Tc2_Mc2.MC_Reset;
	fbMcMoveAbs	: Tc2_Mc2.MC_MoveAbsolute;
	fbMcMoveMod	: Tc2_Mc2.MC_MoveModulo;
	fbMcMoveRel	: Tc2_Mc2.MC_MoveRelative;
	fbMcMoveVel	: Tc2_Mc2.MC_MoveVelocity;

	//rising edge detection
	bExecMove_	: BOOL;
	bExecHWDiag_: BOOL;
	bExecHWRes_	: BOOL;
	bExecReset_	: BOOL;
END_VAR

;

METHOD M_Diag : BOOL
VAR_INPUT
END_VAR
VAR_OUTPUT
	bNcError 	: BOOL;
	bDrvError 	: BOOL;
	iNcErrorId	: UDINT;
END_VAR
//get axis diag
sAxis.ReadStatus();
bNcError	:= sAxis.NcToPlc.StateDWord.31;
bDrvError	:= sAxis.NcToPlc.StateDWord.28;
iNcErrorId	:= sAxis.NcToPlc.ErrorCode;
M_Diag 		:= bNcError OR bDrvError OR (iNcErrorId <> 0);
END_METHOD

METHOD M_Enable : BOOL
VAR_INPUT
	bEnable		: BOOL;
	fOverride	: LREAL;
END_VAR
//enable axis
fbMcPower(
	Enable		:= bEnable, 	Enable_Positive	:= bEnable,	Enable_Negative	:= bEnable, 
	Override	:= fOverride, 	Axis			:= sAxis
);
M_Enable := fbMcPower.Status;
END_METHOD

METHOD M_HardwareDiag : BOOL
VAR_INPUT
	bExecute	: BOOL;
END_VAR
//get hardware diag --> overwrite method if necessary
CASE eCurState OF
eAxisState_Idle:
	IF bExecute AND NOT bExecHWDiag_ THEN
		eCurState := eAxisState_Diag;
	END_IF

eAxisState_Diag:
		eCurState := eAxisState_Idle;

END_CASE

M_HardwareDiag 	:= eCurState <> eAxisState_Idle;	
bExecHWDiag_	:= bExecute;
END_METHOD

METHOD M_HardwareReset : BOOL
VAR_INPUT
	bExecute	: BOOL;
END_VAR
//hardware reset axis --> overwrite method if necessary
CASE eCurState OF
eAxisState_Idle:
	IF bExecute AND NOT bExecHWRes_ THEN
		eCurState := eAxisState_Reset;
	END_IF

eAxisState_Reset:
		eCurState := eAxisState_Idle;

END_CASE

M_HardwareReset := eCurState <> eAxisState_Idle;	
bExecHWRes_		:= bExecute;
END_METHOD

METHOD M_Move : BOOL
VAR_INPUT
	bExecute	: BOOL;
	eMoveCmd	: E_MoveCmd;
	fVelocity	: LREAL;
	fPosition	: LREAL;
END_VAR
//move axis
CASE eCurState OF
eAxisState_Idle:	
	IF bExecute AND NOT bExecMove_ THEN
		CASE eMoveCmd OF
		eCmd_MoveAbsolute:
			fbMcMoveAbs(
				Execute	:= bExecute, 	Position:= fPosition,	Velocity:= fVelocity, 
				Axis	:= sAxis, 		Done	=> bDone,		Busy	=> bBusy, 
				Active	=> bActive, 	Error	=> bError,		ErrorID	=> iErrorId
			);
			eCurState := eAxisState_Move;
		
		eCmd_MoveModulo:
			fbMcMoveMod(
				Execute	:= bExecute, 	Position:= fPosition,	Velocity:= fVelocity, 
				Axis	:= sAxis, 		Done	=> bDone, 		Busy	=> bBusy, 
				Active	=> bActive, 	Error	=> bError,		ErrorID	=> iErrorId
			);
			eCurState := eAxisState_Move;
		
		eCmd_MoveRelative:
			fbMcMoveRel(
				Execute	:= bExecute, 	Distance:= fPosition,	Velocity:= fVelocity, 
				Axis	:= sAxis, 		Done	=> bDone,		Busy	=> bBusy, 
				Active	=> bActive, 	Error	=> bError,		ErrorID	=> iErrorId
			);
			eCurState := eAxisState_Move;
		
		eCmd_MoveVelocity:
			fbMcMoveVel(
				Execute	:= bExecute, 	Velocity:= fVelocity,	Axis	:= sAxis, 
				InVelocity=> bDone,		Busy	=> bBusy,		Active	=> bActive, 
				Error	=> bError, 		ErrorID	=> iErrorId,	Busy	=> bBusy,
				Active	=> bActive,		Error	=> bError,		ErrorID	=> iErrorId
			);		
			eCurState := eAxisState_Move;
		END_CASE
	END_IF
		
eAxisState_Move:
	CASE eMoveCmd OF
	eCmd_MoveAbsolute:
		fbMcMoveAbs(
			Execute	:= TRUE, 		Position:= fPosition,	Velocity:= fVelocity, 
			Axis	:= sAxis, 		Done	=> bDone,		Busy	=> bBusy, 
			Active	=> bActive, 	Error	=> bError, 		ErrorID	=> iErrorId
		);
		IF bDone OR bError THEN
			fbMcMoveAbs(Execute	:= FALSE,Axis := sAxis); 
			eCurState := eAxisState_Idle;
		END_IF
	
	eCmd_MoveModulo:
		fbMcMoveMod(
			Execute	:= TRUE, 		Position:= fPosition,	Velocity:= fVelocity, 
			Axis	:= sAxis, 		Done	=> bDone,		Busy	=> bBusy, 
			Active	=> bActive, 	Error	=> bError,		ErrorID	=> iErrorId
		);
		IF bDone OR bError THEN
			fbMcMoveMod(Execute	:= FALSE,Axis := sAxis); 
			eCurState := eAxisState_Idle;
		END_IF
	
	eCmd_MoveRelative:
		fbMcMoveRel(
			Execute	:= TRUE, 		Distance:= fPosition,	Velocity:= fVelocity, 
			Axis	:= sAxis, 		Done	=> bDone,		Busy	=> bBusy, 
			Active	=> bActive, 	Error	=> bError,		ErrorID	=> iErrorId
		);
		IF bDone OR bError THEN
			fbMcMoveRel(Execute	:= FALSE,Axis := sAxis); 
			eCurState := eAxisState_Idle;
		END_IF
	
	eCmd_MoveVelocity:
		fbMcMoveVel(
			Execute	:= TRUE, 		Velocity:= fVelocity,	Axis	:= sAxis, 
			InVelocity=> bDone,		Busy	=> bBusy,		Active	=> bActive, 
			Error	=> bError, 		ErrorID	=> iErrorId,	Busy	=> bBusy, 		
			Active	=> bActive,		Error	=> bError,		ErrorID	=> iErrorId
		);		
		IF bDone OR bError THEN
			fbMcMoveVel(Execute	:= FALSE,Axis := sAxis); 
			eCurState := eAxisState_Idle;
		END_IF
	END_CASE
END_CASE

M_Move 		:= (eCurState <> eAxisState_Idle);
bExecMove_	:= bExecute;
END_METHOD

METHOD M_Reset : BOOL
VAR_INPUT
	bExecute	: BOOL;
END_VAR
//reset nc axis
CASE eCurState OF
eAxisState_Idle:
	IF bExecute AND NOT bExecReset_ THEN
		fbMcReset(
			Execute	:= bExecute, 	Axis	:= sAxis,	Done	=> bDone, 
			Busy	=> bBusy, 		Error	=> bError,	ErrorID	=> iErrorId 
		);
		eCurState := eAxisState_Reset;
	END_IF

eAxisState_Reset:
	fbMcReset(
		Execute	:= FALSE, 	Axis	:= sAxis,	Done	=> bDone, 
		Busy	=> bBusy, 	Error	=> bError,	ErrorID	=> iErrorId 
	);
	IF fbMcReset.Done OR fbMcReset.Error THEN
		eCurState := eAxisState_Idle;
	END_IF
END_CASE

M_Reset 	:= eCurState <> eAxisState_Idle;	
bExecReset_	:= bExecute;
END_METHOD

END_FUNCTION_BLOCK

// ---- POUs/Sample OOP Conveyor/FB_OOPConveyor.TcPOU
FUNCTION_BLOCK FB_OOPConveyor
VAR_INPUT
	eSampleModeIn		: E_SampleMode;	
END_VAR
VAR_IN_OUT
	AxisRef				: ARRAY [1..iMAX_AXES_REF] OF Tc2_MC2.AXIS_REF;			// axis reference (process data plc/nc)
END_VAR
VAR_OUTPUT
	eSampleModeOut		: E_SampleMode;	
END_VAR
VAR
	iCounter 			: DINT;	

	//axes FB instances
	fbConv1Axis			: FB_AxisNc;
	fbConv2Axis 		: FB_VeryBasicMotor;
	fbConv3Axis 		: FB_AX5000;
	
	//axes interfaces	
	ipConv1Axis 		: I_Axis;
	ipConv2Axis 		: I_Axis;
	ipConv3Axis 		: I_Axis;
	
	//drive references
	stConv3DriveRef 	: ST_DRIVEREF;
	
	//station
	fbStation			: FB_Station;
	fbTransfer1 		: FB_TransferStation;
	fbTransfer2 		: FB_TransferStation;
	
	//conveyor
	fbInfeedConveyor 	: FB_Conveyor;
	fbConveyor2 		: FB_Conveyor;
	fbConveyor3 		: FB_Conveyor;

	//other variables
	bAllowJog			: BOOL;
	bEnableAxis1		: BOOL := TRUE;
	bJogActive			: BOOL;
	eMachineState		: E_Modes := E_SwitchingToAuto;
	iInfeedManualRequest: UDINT;
	bJogBwd AT %I*		: BOOL;
	bJogFwd AT %I*		: BOOL;
	I					: INT;
	fJogSpeed			: LREAL :=200;
	fConveyorCmdSpeed	: LREAL :=10;
	bRunConveyor		: BOOL := TRUE;
	iAnalogValue		: INT;
	bPartPresent		: BOOL;
	iAcceptPartStatus	: UDINT;
	bPickPart			: BOOL;
	iTransferPartStatus	: UDINT;
	fbTrigNewPart		: R_TRIG;
	iTransferPlacePartStatus: UDINT;
	bPlacePart			: BOOL;
	iTransfer2Status	: UDINT;
	bPickPart2			: BOOL;
	bPlacePart2			: BOOL;
	iRemoveFromConveyor3Status: UDINT;
	stOutfeedpart 		: ST_PartData;
	bRemovePart			: BOOL;
	bPartRemoved		: BOOL;
	stEmptyPart			: ST_PartData;
	bBusy				: BOOL;
	Timer				: TON := (PT := T#30s);
END_VAR

iCounter := iCounter + 1;

IF (eSampleModeIn = eSMode_OOPConv_Req) OR (eSampleModeOut = eSMode_OOPConv_Act) THEN
	//call conveyor axes
	fbConv1Axis(stAxisRef := AxisRef[1]); //FB_Axis
	fbConv2Axis(iAnalogInput := iAnalogValue, fScalingFactor:= 1, iAnalogOutput=>iAnalogValue ); //FB_VeryBasicMotor
	fbConv3Axis(stAxisRef := AxisRef[2], stDriveRef:= stConv3DriveRef); //FB_AX5000
	
	//assign axes interfaces
	ipConv1Axis := fbConv1Axis;
	ipConv2Axis := fbConv2Axis;
	ipConv3Axis := fbConv3Axis;
	
	//call conveyor FBs
	fbInfeedConveyor(fbAxis:= ipConv1Axis);
	fbConveyor2(fbAxis := ipConv2Axis);
	fbConveyor3(fbAxis := ipConv3Axis);
	
	//call stations 
	fbTransfer1(fbConveyorToPickFrom:= fbInfeedConveyor , fbConveyorToPlaceTo:= fbConveyor2 , fbStation:= fbStation);
	fbTransfer2(fbConveyorToPickFrom:= fbConveyor2 , fbConveyorToPlaceTo:= fbConveyor3 , fbStation:= fbStation);
	
	//call station
	fbStation();
	CASE eMachineState OF
		E_Disabled: 
			//Machine is disabled
			fbInfeedConveyor.P_DeviceID :=1;
			fbTransfer1.P_DeviceID := 2;
			fbStation.P_DeviceID:= 3;
			fbConveyor2.P_DeviceID := 4;
			fbConveyor3.P_DeviceID := 5;
			fbInfeedConveyor.P_MinimumSpacing := 50;
			fbInfeedConveyor.P_StartLocation := 10;
			fbInfeedConveyor.P_PickLocation := 300;
			fbConveyor2.P_MinimumSpacing:= 75;
			fbConveyor2.P_StartLocation := 10;
			fbConveyor2.P_PickLocation := 200;
			fbConveyor3.P_MinimumSpacing:= 20;
			fbConveyor3.P_StartLocation := 10;
			fbConveyor3.P_PickLocation := 600;
			FOR I := 1 TO 100 DO   
				arrParts[I].fLength := 10;
			END_FOR  
			
		E_Error: 
			;  //Machine is in an error state
			
		E_SwitchingToAuto: 
			//Reqeuest Auto from all devices 
			fbInfeedConveyor.M_Auto(bRequestAutoMode:= TRUE);
			fbStation.M_Auto(bRequestAutoMode:=TRUE );
			fbConveyor2.M_Auto(bRequestAutoMode:= TRUE);
			fbConveyor3.M_Auto(bRequestAutoMode:= TRUE);
			fbTransfer1.M_Auto(bRequestAutoMode:= TRUE);
			
			// If all devices are in auto mode then the machine is in Auto mode
			IF fbInfeedConveyor.P_CurrentState = E_Auto  
			  AND fbStation.P_CurrentState = E_Auto 
			  AND fbConveyor2.P_CurrentState = E_Auto 
			  AND fbTransfer1.P_CurrentState = E_Auto
			  AND fbConveyor3.P_CurrentState = E_Auto THEN 
					eMachineState:= E_Auto;
					fbInfeedConveyor.M_Auto(bRequestAutoMode:= FALSE);
					fbTransfer1.M_Auto(bRequestAutoMode := FALSE);
					fbStation.M_Auto(bRequestAutoMode:=FALSE);
					fbConveyor2.M_Auto(bRequestAutoMode:= FALSE);
					fbConveyor3.M_Auto(bRequestAutoMode:= FALSE);
					
			//If any devices are in Error mode then the machine is in the error state
			ELSIF fbInfeedConveyor.P_CurrentState = E_Error  
			  OR fbStation.P_CurrentState = E_Error 
			  OR fbConveyor2.P_CurrentState = E_Error     
			  OR fbTransfer1.P_CurrentState = E_Error
			  OR fbConveyor3.P_CurrentState = E_Error THEN  
					eMachineState:= E_Error;
					fbTransfer1.M_Auto(bRequestAutoMode := FALSE);
					fbInfeedConveyor.M_Auto(bRequestAutoMode:= FALSE);
					fbStation.M_Auto(bRequestAutoMode:=FALSE );
					fbConveyor2.M_Auto(bRequestAutoMode:= FALSE);
					fbConveyor3.M_Auto(bRequestAutoMode:= FALSE);
			END_IF
			
		E_SwitchingToManual:
			//Reqeuest Manual from all devices 
			fbInfeedConveyor.M_Manual(bRequestManualMode:= TRUE);
			fbStation.M_Manual(bRequestManualMode:= TRUE);
			fbConveyor2.M_Manual(bRequestManualMode:=TRUE );
			fbConveyor3.M_Manual(bRequestManualMode:=TRUE );
			fbTransfer1.M_Manual(bRequestManualMode:=TRUE);
			// If all devices are in Manual mode then the machine is in Manual mode
			IF fbInfeedConveyor.P_CurrentState = E_Manual 
			  AND fbConveyor2.P_CurrentState = E_Manual 
			  AND fbConveyor3.P_CurrentState = E_Manual
			  AND fbTransfer1.P_CurrentState = E_Manual
			  AND fbStation.P_CurrentState = E_Manual  THEN
					eMachineState:= E_Manual;
					fbInfeedConveyor.M_Manual(bRequestManualMode:= FALSE);
					fbStation.M_Manual(bRequestManualMode:= FALSE);
					fbConveyor2.M_Manual(bRequestManualMode:=FALSE );
					fbTransfer1.M_Manual(bRequestManualMode:=FALSE);
					fbConveyor3.M_Manual(bRequestManualMode:=FALSE);
			//If any devices are in Error mode then the machine is in the error state
			ELSIF fbInfeedConveyor.P_CurrentState = E_Error 
			  OR fbConveyor2.P_CurrentState = E_Error 
			  OR fbConveyor3.P_CurrentState = E_Error
			  OR fbTransfer1.P_CurrentState = E_Error
			  OR  fbStation.P_CurrentState = E_Error THEN 
					eMachineState:= E_Error;
					fbInfeedConveyor.M_Manual(bRequestManualMode:= FALSE);
					fbStation.M_Manual(bRequestManualMode:= FALSE);
					fbTransfer1.M_Manual(bRequestManualMode:=FALSE);
					fbConveyor2.M_Manual(bRequestManualMode:=FALSE );
					fbConveyor3.M_Manual(bRequestManualMode:=FALSE);
			END_IF
		
		E_Resetting: 
			fbInfeedConveyor.M_Reset(bRequestReset:=TRUE );
			fbConveyor2.M_Reset(bRequestReset:=TRUE);
			fbConveyor3.M_Reset(bRequestReset:=TRUE);
			fbStation.M_Reset(bRequestReset:= TRUE);
			IF fbInfeedConveyor.P_CurrentState = E_Reset 
			  AND fbConveyor2.P_CurrentState = E_Reset 
			  AND fbConveyor3.P_CurrentState = E_Reset
			  AND fbStation.P_CurrentState = E_Reset THEN
				eMachineState := E_Reset;
				fbInfeedConveyor.M_Reset(bRequestReset:=FALSE );
				fbConveyor2.M_Reset(bRequestReset:=FALSE);
				fbConveyor3.M_Reset(bRequestReset:=FALSE);
				fbStation.M_Reset(bRequestReset:= FALSE);
			ELSIF fbInfeedConveyor.P_CurrentState = E_Error   
			  OR fbConveyor2.P_CurrentState = E_Error 
			  OR fbConveyor3.P_CurrentState = E_Error
			  OR  fbStation.P_CurrentState = E_Error THEN 
					eMachineState:= E_Error;
					fbInfeedConveyor.M_Reset(bRequestReset:=FALSE );
					fbConveyor2.M_Reset(bRequestReset:=FALSE);
					fbConveyor3.M_Reset(bRequestReset:=FALSE);
					fbStation.M_Reset(bRequestReset:= FALSE);
			END_IF
		
		E_Reset: 
			// Machine has been reset and awaits a mode change to Manual or Auto
			 ;
	
							
		E_Manual :  
			// Manual Mode allow all manual commands
			fbInfeedConveyor.bJogConveyorFwd:=bJogFwd; 
			fbInfeedConveyor.bJogConveyorBwd:=bJogBwd; 
			fbInfeedConveyor.fJogSpeed:= fJogSpeed;
			fbConveyor2.fJogSpeed:=fJogSpeed;
			fbConveyor2.bJogConveyorFwd:=bJogFwd; 
			fbConveyor2.bJogConveyorBwd:=bJogBwd;
			fbConveyor3.bJogConveyorFwd:=bJogFwd;
			fbConveyor3.bJogConveyorBwd:=bJogBwd; 
			fbConveyor3.fJogSpeed:=fJogSpeed;
			
		E_Auto :		
			fbInfeedConveyor.fCmdSpeed:= fConveyorCmdSpeed;
			fbInfeedConveyor.bRunConveyor := bRunConveyor;
			fbConveyor2.bRunConveyor := bRunConveyor;
			fbConveyor2.fCmdSpeed := fConveyorCmdSpeed +5;
			fbConveyor3.bRunConveyor := bRunConveyor;
			fbConveyor3.fCmdSpeed := fConveyorCmdSpeed +3;
			//button triggers a part is presetn
			fbTrigNewPart(CLK:= bPartPresent);
			IF fbTrigNewPart.Q THEN 
				arrParts[1].iIDNumber:= arrParts[1].iIDNumber + 5 ;
			END_IF
			iAcceptPartStatus := fbInfeedConveyor.M_AcceptPart(bPartPresentAtEntrance:=bPartPresent , stPartAtEntrance:=arrParts[1] );
			//Part has been accepted by conveyor 
			IF iAcceptPartStatus = 3 THEN 
				bPartPresent := FALSE;
			END_IF
			iTransferPartStatus := fbTransfer1.M_PickPart(bGetPart:=bPickPart, bPartAvailable := fbInfeedConveyor.bPartInPickLocation );
			IF  bPlacePart (*fbTransfer1.bHavePart*) THEN 
				iTransferPlacePartStatus := fbTransfer1.M_PlacePart(bPlacePart:=TRUE );
			END_IF
			iTransfer2Status := fbTransfer2.M_PickPart(bGetPart:=bPickPart2, bPartAvailable := fbConveyor2.bPartInPickLocation );
			IF  bPlacePart2 (*fbTransfer1.bHavePart*) THEN 
				iTransfer2Status := fbTransfer2.M_PlacePart(bPlacePart:=TRUE);
			END_IF
	
			IF fbConveyor3.bPartInPickLocation THEN 
				bRemovePart := TRUE;
			END_IF
			IF stOutfeedpart.iIDNumber <>0 THEN 
				bPartRemoved := TRUE; 
			END_IF 	
			iRemoveFromConveyor3Status := fbConveyor3.M_ReleasePart(bReleasePartReq:=bRemovePart , bPartHandedOff:=bPartRemoved , stPartToRelease=>stOutfeedpart );
			IF iRemoveFromConveyor3Status = 3 THEN 
				stOutfeedpart := stEmptyPart;
				bRemovePart:=FALSE;
				bPartRemoved := FALSE;
			END_IF	
			
	END_CASE

	Timer(IN := TRUE);
	IF Timer.Q THEN
		Timer(IN := FALSE);
		bBusy := FALSE;
	ELSE
		bBusy := TRUE;
	END_IF
	
	IF bBusy THEN
		eSampleModeOut := eSMode_OOPConv_Act;
	ELSE
		eSampleModeOut := eSMode_Idle;
	END_IF
END_IF

END_FUNCTION_BLOCK

// ---- POUs/Sample OOP Conveyor/Axis Blocks/FB_AxisNc.TcPOU
FUNCTION_BLOCK FB_AxisNc IMPLEMENTS I_Axis
VAR_INPUT
END_VAR
VAR_OUTPUT
END_VAR
VAR_IN_OUT
	stAxisRef 		: Tc2_MC2.AXIS_REF;
END_VAR
VAR
//Enable	
	fbMCPower		: Tc2_MC2.MC_Power;
	bEnableAxis		: BOOL;
	fbTrigEnable	: R_TRIG;
	
//Jog	
	fbJog			: Tc2_MC2.MC_Jog;
	bJogAxisFwd		: BOOL;
	bJogAxisBwd		: BOOL;
	fJogAxisSpeed	: LREAL;
	fbJogErrTrig	: R_TRIG;
	bJogError		: BOOL;
	udiJogErrID		: UDINT;
	
//Move Velocity 	
	fbMoveVelocity 	: Tc2_MC2.MC_MoveVelocity;
	eAxisDirection	: Tc2_MC2.MC_Direction;
	fbStartMoveVelocity: R_TRIG;
	iVeloMoveSeq	: INT;
	
//Reset	
	fbMCReset		: Tc2_MC2.MC_Reset;
	fbTrigResetSeq	: R_TRIG;
	iResetSeq		: INT;
	bError			: BOOL;
	udiErrorID		: UDINT;
	fbTrigStop		: R_TRIG;
	iStopSeq		: INT;
	fbMCStop		: Tc2_MC2.MC_Stop;
END_VAR

stAxisRef.ReadStatus();

//the MC_Power block is one that should be called every cycle to allow for a very quick disabling of the axis
fbMCPower(
	Enable			:= bEnableAxis , 
	Enable_Positive	:= bEnableAxis , 
	Enable_Negative	:= bEnableAxis , 
	Override		:= 100.0 , 
	Axis			:= stAxisRef );

METHOD M_Disable : UDINT
VAR_INPUT
	bDisable : BOOL;
END_VAR
//The result of the method is an unsigned double integer
// 0 = idle 
// 1 = busy
// 3 = complete
// Any other number = Error
IF NOT bDisable THEN
	M_Disable := 0;
END_IF

IF bDisable THEN 
	bEnableAxis := FALSE;
	M_Disable := 1;
END_IF

IF NOT fbMCPower.Status THEN
	M_Disable := 3;
END_IF
END_METHOD

METHOD M_Enable : UDINT
VAR_INPUT
	bEnable : BOOL;
END_VAR
//The result of the method is an unsigned double integer
// 0 = idle 
// 1 = busy
// 3 = complete
// Any other number = Error
IF bEnable THEN
	bEnableAxis := TRUE;
	M_Enable := 1;
END_IF

IF fbMCPower.Status THEN
	M_Enable := 3;
END_IF

IF fbMCPower.Error THEN
	M_Enable :=fbMCPower.ErrorID;
END_IF

IF NOT bEnable THEN
	M_Enable := 0;
END_IF
END_METHOD

METHOD M_HardwareReset : UDINT
VAR_INPUT
	bReset	: BOOL;
END_VAR
//The result of the method is an unsigned double integer
// 0 = idle 
// 1 = busy
// 3 = complete
// Any other number = Error
// Default result for the method is that it completes
IF bReset THEN
	M_HardwareReset := 3;
END_IF

IF NOT bReset THEN
	M_HardwareReset := 0;
END_IF
END_METHOD

METHOD M_Jog : UDINT
VAR_INPUT
	bJogFwd 	: BOOL;
	bJogBwd 	: BOOL;
	fJogSpeed 	: LREAL;
END_VAR
//The result of the method is an unsigned double integer
// 0 = idle 
// 1 = busy
// 3 = complete
// Any other number = Error
IF bJogFwd AND NOT bJogBwd THEN
	bJogAxisFwd := TRUE;
	bJogAxisBwd := FALSE;
ELSIF bJogBwd AND NOT bJogFwd THEN
	bJogAxisBwd := TRUE;
	bJogAxisFwd := FALSE;
ELSE
	bJogAxisBwd := FALSE;
	bJogAxisFwd := FALSE;
END_IF

fbJog(
	JogForward	:= bJogAxisFwd, 
	JogBackwards:= bJogAxisBwd, 
	Velocity	:= fJogSpeed, 
	Mode 		:= MC_JOGMODE_CONTINOUS,
	Axis		:= stAxisRef
);
	
fbJogErrTrig(CLK := fbJog.Error);
IF fbJogErrTrig.Q THEN
	bJogError:=TRUE;
	udiJogErrID := fbJog.ErrorID;
END_IF

IF fbJog.Active THEN
	M_Jog := 1;
ELSIF fbJog.Error THEN
	M_Jog := fbJog.ErrorID;
ELSE
	M_Jog := 0;
END_IF
END_METHOD

METHOD M_Reset : UDINT
VAR_INPUT
	bReset : BOOL;
END_VAR
//The result of the method is an unsigned double integer
// 0 = idle 
// 1 = busy
// 3 = complete
// Any other number = Error
VAR
	udiHardwareResetResult:UDINT;
END_VAR
fbTrigResetSeq(CLK:=bReset);
IF fbTrigResetSeq.Q THEN
	M_Reset		:= 1;
	iResetSeq	:= 10;
END_IF

IF NOT bReset THEN
	M_Reset 	:= 0;
END_IF

CASE iResetSeq OF 
	0: (* Idle*)
		fbMCReset(Execute := FALSE, Axis := stAxisRef);
		
	10: (*If necessary reset the hardware first*)
		M_HardwareReset(bReset:=TRUE);
		iResetSeq := 10;	
	20: 
		udiHardwareResetResult := M_HardwareReset(bReset:=TRUE);   
		IF udiHardwareResetResult = 3 THEN // Hardware reset successful
			M_HardwareReset(bReset:=FALSE);
			iResetSeq := 30;
		ELSIF udiHardwareResetResult > 3 THEN // Hardware reset faulted
			M_Reset := udiHardwareResetResult;
			iResetSeq:= 0;			
		END_IF
		fbMCReset(Execute:=TRUE ,Axis:= stAxisRef);
		iResetSeq := 30;
	30:
		fbMCReset(Axis:=stAxisRef);
		IF fbMCReset.Done OR fbMCReset.Error THEN
			fbMCReset(Execute:=FALSE,Axis:=stAxisRef);
			iResetSeq := 0;
			IF fbMCReset.Error THEN
				M_Reset := fbMCReset.ErrorID;
			ELSE
				iResetSeq:= 0;		
				M_Reset:=2;
			END_IF
		END_IF
END_CASE
END_METHOD

METHOD M_Speed : UDINT
VAR_INPUT
	bMoveVelocity 	: BOOL;
	fSpeed 			: LREAL;
END_VAR
//The result of the method is an unsigned double integer
// 0 = idle 
// 1 = busy
// 3 = complete
// Any other number = Error
//Determine the dirction of the velocity command
IF fSpeed > 0 THEN
	eAxisDirection := MC_Positive_Direction; 
ELSE
	eAxisDirection := MC_Negative_Direction;
END_IF
//Look for a trigger 
fbStartMoveVelocity(CLK:= bMoveVelocity);
IF fbStartMoveVelocity.Q THEN 
	iVeloMoveSeq := 10;
	M_Speed:=1;
	fbMoveVelocity(Execute:= FALSE,Axis:=stAxisRef);
END_IF
// If the bMoveVelocity bit is off clear the Method
IF NOT bMoveVelocity THEN
	M_Speed := 0;
END_IF

CASE iVeloMoveSeq OF
	0: (*Idle*)
		fbMoveVelocity(Execute:=FALSE,Axis:=stAxisRef);
	10: (*Initiate Move Velocity command*)
		fbMoveVelocity(
			Execute:= TRUE , 
			Velocity:= ABS(fSpeed), 
			Direction:= eAxisDirection , 
			Axis:=stAxisRef);
		iVeloMoveSeq := 20;
		
	20: (*Wait for axis to reach velocity or error out*)
		fbMoveVelocity(Axis:=stAxisRef);
		IF fbMoveVelocity.InVelocity OR fbMoveVelocity.Error THEN
			IF fbMoveVelocity.Error THEN
				M_Speed := fbMoveVelocity.ErrorID;
			END_IF			
			fbMoveVelocity(Execute:= FALSE,Axis:=stAxisRef);
			iVeloMoveSeq:=0;
			M_Speed:=3;
		END_IF
END_CASE
END_METHOD

METHOD M_Stop : UDINT
VAR_INPUT
	bStop	: BOOL;
END_VAR
//The result of the method is an unsigned double integer
// 0 = idle 
// 1 = busy
// 3 = complete
// Any other number = Error
VAR

END_VAR
//Look for a trigger 
fbTrigStop(CLK:= bStop);
IF fbTrigStop.Q THEN 
	iStopSeq := 10;
	M_Stop:=1;
END_IF
// If the bMoveVelocity bit is off clear the Method
IF NOT bStop THEN
	M_Stop := 0;
END_IF

CASE iStopSeq OF
	0: (*Idle*)
		fbMCStop(Execute:=FALSE,Axis:=stAxisRef);
	10: (*Initiate Move Velocity command*)
		fbMCStop(Execute:= TRUE,Axis:=stAxisRef);
		iStopSeq := 20;
		
	20: (*Wait for axis to reach velocity or error out*)
		fbMCStop(Axis:=stAxisRef);
		IF fbMCStop.Done OR fbMCStop.Error THEN
			IF fbMCStop.Error THEN
				M_Stop := fbMCStop.ErrorID;
			END_IF			
			fbMCStop(Execute:= FALSE,Axis:=stAxisRef);
			iStopSeq:=0;
			M_Stop:=3;
		END_IF
END_CASE
END_METHOD

PROPERTY P_CurrentPosition : LREAL
GET
P_CurrentPosition :=  stAxisRef.NcToPlc.ActPos;
END_GET
SET
END_SET
END_PROPERTY

PROPERTY P_CurrentSpeed : LREAL
GET
P_CurrentSpeed := stAxisRef.NcToPlc.ActVelo;
END_GET
SET
// setting the current speed is not allowed
;
END_SET
END_PROPERTY

PROPERTY P_Error : BOOL
GET
//Report Errors with the most important first 
// Axis Hardware Failure
// NC Axis Failure
//Move command errors are returned by their respective method calls
P_Error := stAxisRef.Status.Error;
END_GET
SET
//Allow user to externally clear error.
IF P_Error = FALSE THEN
	udiErrorID	:= 0;
	bError 		:= FALSE;
END_IF
END_SET
END_PROPERTY

PROPERTY P_ErrorID : UDINT
GET
P_ErrorID := udiErrorID;
END_GET
SET
IF P_ErrorID = 0 THEN
	bError		:= FALSE;
	udiErrorID	:= 0;
END_IF
END_SET
END_PROPERTY

PROPERTY P_Ready : BOOL
GET
IF stAxisRef.Status.ControlLoopClosed AND NOT stAxisRef.Status.Error THEN
	P_Ready := TRUE;
ELSE
	P_Ready := FALSE;
END_IF
END_GET
SET
;
END_SET
END_PROPERTY

END_FUNCTION_BLOCK

// ---- POUs/Motion/Axis1.TcPOU
PROGRAM Axis1
VAR

	sAxisDescription						:STRING	:= 'Axis 1 - EL7037 - AS1020-0120';	

(* Axis - basic functions *)
	fbAxis									:FB_Axis;
	fMoveAbsPosition						:LREAL;				(* Target position *)
	fMoveAbsVelocity						:LREAL	:= 500.0;	(* Target speed axis 1 max. 3600.0 Degree/s *)
	bStartMoveAbs							:BOOL;
	bMoveAbsBusy							:BOOL;
	bMoveAbsDone							:BOOL;
	bAxisErr								:BOOL;
	nAxisErrId								:DWORD;
	bReset									:BOOL;
	bStop									:BOOL;
	bStopAxisDone							:BOOL;
	bStopAxisBusy							:BOOL;
	bRevSeqStart							:BOOL;
	bStartparameterSet						:BOOL;
	
(* Test - change target position *)
	bTestChangeTargetPos					:BOOL;				(* Test - change target position *)
	bMaxPositionReached						:BOOL;
	
(* Homing *)
	fbHomingAxis							:Tc2_Mc2.MC_Home;
	fHomingPosition							:LREAL	:= 331.00;

(* Touch Probe *)
	fbTouchProbe							:Tc2_Mc2.MC_TouchProbe;
	stTriggerInput							:Tc2_Mc2.TRIGGER_REF;
	bTouchProbeDone							:BOOL;
	bTouchProbeBusy							:BOOL;
	bTouchProbeComAb						:BOOL;
	bTouchProbeErr							:BOOL;
	bTouchProbeErrId						:UDINT;
	fRecordedPosition 						:LREAL;
	stRecordedData							:MC_TouchProbeRecordedData;	

(* Couple Axis on Handwheel *)
	fbGearIn								:Tc2_Mc2.MC_GearIn;
	bGearInDone								:BOOL;
	bAxisCoupled							:BOOL;

(* Uncouple Axis *)
	fbGearOut								:Tc2_Mc2.MC_GearOut;
	bGearOutDone							:BOOL;

END_VAR
(* End *)

(* Axis 1 *)

(* Axis - basic functions  *)

	IF NOT bStartparameterSet
	THEN
		(* Startup Parameter reversing sequence *)
		fbAxis.fRevSeqTargetPos1	:= 720.0;
		fbAxis.fRevSeqTargetVelo1	:= 500.0;
		fbAxis.fRevSeqTargetPos2	:= 0.0;
		fbAxis.fRevSeqTargetVelo2	:= 3000.0;
		fbAxis.nRevSeqIdleTime		:= 500;
		bStartparameterSet			:= TRUE;
	END_IF
		
	fbAxis(
		bPowerEnable		:= 	bSwitchS12,
		fPowerOverride		:= 	F_Scaling(nAnalogInR10, 100.0, 32767.0),
		bMoveAbsExecute		:= 	(bStartMoveAbs OR bSwitchS16) AND NOT stAxis1.Status.Coupled,
		fMoveAbsPosition	:= 	fMoveAbsPosition,
		fMoveAbsVelocity	:= 	fMoveAbsVelocity,
		bReset				:= 	bReset OR bSwitchS21,
		bStopAxis			:= 	bStop,
		bRevSeqStart		:=  (bSwitchS20 OR bRevSeqStart) AND fbAxis.bPowerStatus, 
		stAxis				:= 	stAxis1,
		bPowerStatus		=> 	bLedH12,
		bMoveAbsDone		=> 	bMoveAbsDone,
		bMoveAbsBusy		=> 	bMoveAbsBusy,
		bAxisErr			=> 	bAxisErr,
		nAxisErrId			=> 	nAxisErrId,
		bStopAxisDone		=> 	bStopAxisDone,
		bStopAxisBusy		=> 	bStopAxisBusy);
		

(* Test - change target position - Axis *)
	IF bTestChangeTargetPos
		AND (fMoveAbsPosition <= stAxis1.NcToPlc.ActPos)
			AND NOT bMaxPositionReached
	THEN
		fMoveAbsPosition := fMoveAbsPosition + 180.0;
	ELSE
		IF bTestChangeTargetPos
			AND (fMoveAbsPosition >= 3600.0)
		THEN
			fMoveAbsPosition 	:= 0.0;
			bMaxPositionReached	:= TRUE;
		END_IF
	END_IF

	IF bTestChangeTargetPos
		AND (stAxis1.NcToPlc.ActPos < 1.0)
	THEN
		bMaxPositionReached	:= FALSE;
	END_IF

	IF bSwitchS17
	THEN
		bMaxPositionReached	:= FALSE;
		fMoveAbsPosition 	:= 0.0;
	END_IF
	
(* Homing Axis *)
	fbHomingAxis(
		Execute			:= 	bSwitchS23 AND fbAxis.bPowerStatus,
		Position		:= 	fHomingPosition,
		HomingMode		:= 	MC_DefaultHoming,
		BufferMode		:= 	,
		Options			:= 	,
		bCalibrationCam	:= 	bStepperReferenceCam,
		Axis			:= 	stAxis1,
		Done			=> 	,
		Busy			=> 	,
		Active			=> 	,
		CommandAborted	=> 	,
		Error			=> 	,
		ErrorID			=> 	);
		
		
	bLedH23 :=	(bClock1s 
					AND NOT stAxis1.Status.Homed
					AND fbAxis.bPowerStatus
					AND NOT fbHomingAxis.Busy)
				OR (bClock500ms 
					AND fbHomingAxis.Busy)
				OR fbHomingAxis.Done;
					

(* Touch Probe *)
	stTriggerInput.EncoderID 		:= 1;
	stTriggerInput.TouchProbe 		:= TouchProbe1;
	stTriggerInput.SignalSource 	:= SignalSource_Default;
	stTriggerInput.Edge 			:= RisingEdge;
	stTriggerInput.Mode 			:= TOUCHPROBEMODE_SINGLE;
	stTriggerInput.ModuloPositions 	:= FALSE;

	fbTouchProbe(
		Execute			:= 	bSwitchS24,
		WindowOnly		:= 	,
		FirstPosition	:= 	,
		LastPosition	:= 	,
		Axis			:= 	stAxis1,
		TriggerInput	:= 	stTriggerInput,
		Done			=> 	bTouchProbeDone,
		Busy			=> 	bTouchProbeBusy,
		CommandAborted	=> 	bTouchProbeComAb,
		Error			=> 	bTouchProbeErr,
		ErrorID			=> 	bTouchProbeErrId,
		RecordedPosition=> 	fRecordedPosition,
		RecordedData	=>	stRecordedData);
	
	bLedH24 :=	(bClock500ms 
					AND fbTouchProbe.Busy)
						OR fbTouchProbe.Done;

(* Couple Axis on Handwheel *)
	fbGearIn(
		Execute			:= 	bHandwheelSwitchS28,
		RatioNumerator	:= 	1,
		RatioDenominator:= 	1,
		Acceleration	:= 	,
		Deceleration	:= 	,
		Jerk			:= 	,
		BufferMode		:= 	,
		Options			:= 	,
		Master			:= 	stAxis5,
		Slave			:= 	stAxis1,
		InGear			=> 	bGearInDone,
		Busy			=> 	,
		Active			=> 	,
		CommandAborted	=> 	,
		Error			=> 	,
		ErrorID			=> 	);

(* Axis coupled *)
	bAxisCoupled := stAxis1.Status.Coupled;

(* Uncouple Axis *)
	fbGearOut(
		Execute	:= 	bSwitchS17,
		Options	:= 	,
		Slave	:= 	stAxis1,
		Done	=> 	bGearOutDone,
		Busy	=> 	,
		Error	=> 	,
		ErrorID	=> 	);
	
(* End *)

END_PROGRAM

// ---- POUs/Motion/Components/FB_Axis.TcPOU
FUNCTION_BLOCK FB_Axis
VAR_INPUT
	
	bPowerEnable							:BOOL;
	fPowerOverride							:LREAL;
	bMoveAbsExecute							:BOOL;
	fMoveAbsPosition						:LREAL;
	fMoveAbsVelocity						:LREAL;
	bReset									:BOOL;
	bStopAxis								:BOOL;
	bRevSeqStart							:BOOL;
	bRevSeqStop								:BOOL;
	fRevSeqTargetPos1						:LREAL; 
	fRevSeqTargetVelo1						:LREAL;	 
	fRevSeqTargetPos2						:LREAL;	 
	fRevSeqTargetVelo2						:LREAL; 
	nRevSeqIdleTime							:UINT;
	
END_VAR
VAR_OUTPUT

	bPowerStatus							:BOOL;
	bMoveAbsDone							:BOOL;
	bMoveAbsBusy							:BOOL;
	bAxisErr								:BOOL;
	nAxisErrId								:DWORD;
	bStopAxisDone							:BOOL;
	bStopAxisBusy							:BOOL;
	bRevSeqDone								:BOOL;
	bRevSeqBusy								:BOOL;
	
END_VAR
VAR_IN_OUT

	stAxis									:Tc2_MC2.Axis_Ref;

END_VAR
VAR

	fbMcPower								:Tc2_MC2.MC_Power;
	fbMoveAbsolute							:Tc2_MC2.MC_MoveAbsolute;
	fbReadAxisError							:Tc2_MC2.MC_ReadAxisError;
	fbReset									:Tc2_MC2.MC_Reset;
	fbStop									:Tc2_MC2.MC_Stop;
	fbReversingSequence						:FB_ReversingSequence;

END_VAR
(* End *)

(* FB_Axis *)

(* Read status of the axis *)
	stAxis.ReadStatus();

(* Enable axis *)
	fbMcPower(
		Enable			:= 	bPowerEnable,
		Enable_Positive	:= 	bPowerEnable,
		Enable_Negative	:= 	bPowerEnable,
		Override		:= 	fPowerOverride,
		Axis			:= 	stAxis,
		Status			=> 	bPowerStatus);

(* Start axis at an absolute position *)
	fbMoveAbsolute(
		Execute		:=	bMoveAbsExecute,
		Position	:=	fMoveAbsPosition,
		Velocity	:=	fMoveAbsVelocity,
		Axis		:=	stAxis,
		Done		=>	bMoveAbsDone,
		Busy		=>	bMoveAbsBusy);

(* Read the error code of the axis *)
	fbReadAxisError(
		Enable		:=	TRUE,
		Axis		:=	stAxis,
		AxisErrorID	=>	nAxisErrId);
		
	bAxisErr := nAxisErrId <> 0;

(* Reset axis in case of failure *)
	fbReset(
		Execute		:= 	bReset,
		Axis		:= 	stAxis);

(* Stop axis *)
	fbStop(
		Execute 	:=	bStopAxis,
		Axis		:=	stAxis,
		Done		=>	bStopAxisDone,
		Busy		=>	bStopAxisBusy);

(* Axis reversing sequence *)	
	fbReversingSequence(
		bStart				:= 	bRevSeqStart,
		bStop				:= 	bRevSeqStop,
		fTargetPosition1	:= 	fRevSeqTargetPos1,
		fTargetVelocity1	:= 	fRevSeqTargetVelo1,
		fTargetPosition2	:= 	fRevSeqTargetPos2,
		fTargetVelocity2	:= 	fRevSeqTargetVelo2,
		tIdleTime			:= 	TO_TIME(nRevSeqIdleTime),
		bDone				=> 	bRevSeqDone,
		bBusy				=> 	bRevSeqBusy,
		bErr				=> 	,
		nErrID				=> 	,
		stAxis				:= 	stAxis);
		
(* End *)

END_FUNCTION_BLOCK

// ---- POUs/Motion/Components/FB_ReversingSequence.TcPOU
FUNCTION_BLOCK FB_ReversingSequence
VAR_INPUT
	
	bStart									:BOOL;
	bStop									:BOOL;	
	fTargetPosition1						:LREAL;
	fTargetVelocity1						:LREAL;
	fTargetPosition2						:LREAL;
	fTargetVelocity2						:LREAL;
	tIdleTime								:TIME;
	
END_VAR
VAR_OUTPUT
	
